LIN {X 0,Y 425.386,Z 292.31,A -85,B 0,C 180,E1 -9710.49,E2 -9710.49} C_VEL
LIN {X 0,Y 425.466,Z 292.296,A -85,B 0,C 180,E1 -9713.36,E2 -9713.36} C_VEL
LIN {X 0,Y 425.334,Z 292.312,A -85,B 0,C 180,E1 -9715.261,E2 -9715.261} C_VEL
LIN {X 0,Y 425.553,Z 292.292,A -85,B 0,C 180,E1 -9718.107,E2 -9718.107} C_VEL
LIN {X 0,Y 425.561,Z 292.291,A -85,B 0,C 180,E1 -9720,E2 -9720} C_VEL
LIN {X 0,Y 425.5,Z 292.291,A -85,B 0,C 180,E1 -9722.84,E2 -9722.84} C_VEL
LIN {X 0,Y 425.514,Z 292.294,A -85,B 0,C 180,E1 -9725.687,E2 -9725.687} C_VEL
LIN {X 0,Y 425.384,Z 292.306,A -85,B 0,C 180,E1 -9728.551,E2 -9728.551} C_VEL
LIN {X 0,Y 425.398,Z 292.305,A -85,B 0,C 180,E1 -9732.402,E2 -9732.402} C_VEL
LIN {X 0,Y 425.292,Z 292.321,A -85,B 0,C 180,E1 -9735.331,E2 -9735.331} C_VEL
LIN {X 0,Y 425.302,Z 292.316,A -85,B 0,C 180,E1 -9738.299,E2 -9738.299} C_VEL
LIN {X 0,Y 425.277,Z 292.324,A -85,B 0,C 180,E1 -9741.319,E2 -9741.319} C_VEL
LIN {X 0,Y 425.288,Z 292.318,A -85,B 0,C 180,E1 -9744.651,E2 -9744.651} C_VEL
LIN {X 0,Y 425.238,Z 292.328,A -85,B 0,C 180,E1 -9747.565,E2 -9747.565} C_VEL
LIN {X 0,Y 425.28,Z 292.321,A -85,B 0,C 180,E1 -9750.761,E2 -9750.761} C_VEL
LIN {X 0,Y 425.283,Z 292.318,A -85,B 0,C 180,E1 -9754.284,E2 -9754.284} C_VEL
LIN {X 0,Y 425.268,Z 292.321,A -85,B 0,C 180,E1 -9757.695,E2 -9757.695} C_VEL
LIN {X 0,Y 425.236,Z 292.326,A -85,B 0,C 180,E1 -9760.515,E2 -9760.515} C_VEL
LIN {X 0,Y 425.239,Z 292.326,A -85,B 0,C 180,E1 -9763.35,E2 -9763.35} C_VEL
LIN {X 0,Y 425.251,Z 292.323,A -85,B 0,C 180,E1 -9766.044,E2 -9766.044} C_VEL
LIN {X 0,Y 425.242,Z 292.329,A -85,B 0,C 180,E1 -9768.619,E2 -9768.619} C_VEL
LIN {X 0,Y 425.272,Z 292.323,A -85,B 0,C 180,E1 -9771.1,E2 -9771.1} C_VEL
LIN {X 0,Y 425.29,Z 292.325,A -85,B 0,C 180,E1 -9774.664,E2 -9774.664} C_VEL
LIN {X 0,Y 425.258,Z 292.323,A -85,B 0,C 180,E1 -9778.073,E2 -9778.073} C_VEL
LIN {X 0,Y 425.293,Z 292.317,A -85,B 0,C 180,E1 -9781.366,E2 -9781.366} C_VEL
LIN {X 0,Y 425.257,Z 292.329,A -85,B 0,C 180,E1 -9784.553,E2 -9784.553} C_VEL
LIN {X 0,Y 425.389,Z 292.538,A -85,B 0,C 180,E1 -9787.296,E2 -9787.296} C_VEL
LIN {X 0,Y 426.425,Z 299.768,A -85,B 0,C 180,E1 -9789.247,E2 -9789.247} C_VEL
LIN {X 0,Y 426.191,Z 307.575,A -85,B 0,C 180,E1 -9791.243,E2 -9791.243} C_VEL
LIN {X 0,Y 425.59,Z 319.286,A -85,B 0,C 180,E1 -9794.189,E2 -9794.189} C_VEL
LIN {X 0,Y 425.42,Z 323.878,A -85,B 0,C 180,E1 -9795.256,E2 -9795.256} C_VEL
LIN {X 0,Y 427.716,Z 338.164,A -85,B 0,C 180,E1 -9795.613,E2 -9795.613} C_VEL
LIN {X 0,Y 428.197,Z 343.55,A -85,B 0,C 180,E1 -9795.721,E2 -9795.721} C_VEL
LIN {X 0,Y 427.792,Z 399.196,A -85,B 0,C 180,E1 -9796.671,E2 -9796.671} C_VEL
LIN {X 0,Y 427.517,Z 408.492,A -85,B 0,C 180,E1 -9796.936,E2 -9796.936} C_VEL
LIN {X 0,Y 427.221,Z 418.151,A -85,B 0,C 180,E1 -9797.35,E2 -9797.35} C_VEL
LIN {X 0,Y 426.799,Z 427.305,A -85,B 0,C 180,E1 -9797.881,E2 -9797.881} C_VEL
LIN {X 0,Y 426.301,Z 438.098,A -85,B 0,C 180,E1 -9798.711,E2 -9798.711} C_VEL
LIN {X 0,Y 425.785,Z 447.393,A -85,B 0,C 180,E1 -9799.659,E2 -9799.659} C_VEL
LIN {X 0,Y 425.404,Z 454.053,A -85,B 0,C 180,E1 -9800.491,E2 -9800.491} C_VEL
LIN {X 0,Y 425.02,Z 460.372,A -85,B 0,C 180,E1 -9801.442,E2 -9801.442} C_VEL
LIN {X 0,Y 424.765,Z 465.622,A -85,B 0,C 180,E1 -9802.394,E2 -9802.394} C_VEL
LIN {X 0,Y 424.579,Z 469.999,A -85,B 0,C 180,E1 -9803.346,E2 -9803.346} C_VEL
LIN {X 0,Y 424.42,Z 473.64,A -85,B 0,C 180,E1 -9804.298,E2 -9804.298} C_VEL
LIN {X 0,Y 424.265,Z 476.628,A -85,B 0,C 180,E1 -9805.249,E2 -9805.249} C_VEL
LIN {X 0,Y 424.159,Z 478.944,A -85,B 0,C 180,E1 -9806.2,E2 -9806.2} C_VEL
LIN {X 0,Y 424.151,Z 480.684,A -85,B 0,C 180,E1 -9807.151,E2 -9807.151} C_VEL
LIN {X 0,Y 424.129,Z 481.93,A -85,B 0,C 180,E1 -9808.101,E2 -9808.101} C_VEL
LIN {X 0,Y 424.067,Z 482.706,A -85,B 0,C 180,E1 -9809.05,E2 -9809.05} C_VEL
LIN {X 0,Y 424.039,Z 483,A -85,B 0,C 180,E1 -9810,E2 -9810} C_VEL
LIN {X 0,Y 424.067,Z 482.704,A -85,B 0,C 180,E1 -9810.95,E2 -9810.95} C_VEL
LIN {X 0,Y 424.129,Z 481.925,A -85,B 0,C 180,E1 -9811.899,E2 -9811.899} C_VEL
LIN {X 0,Y 424.15,Z 480.675,A -85,B 0,C 180,E1 -9812.849,E2 -9812.849} C_VEL
LIN {X 0,Y 424.198,Z 477.78,A -85,B 0,C 180,E1 -9814.276,E2 -9814.276} C_VEL
LIN {X 0,Y 424.364,Z 475.142,A -85,B 0,C 180,E1 -9815.226,E2 -9815.226} C_VEL
LIN {X 0,Y 424.496,Z 471.301,A -85,B 0,C 180,E1 -9816.324,E2 -9816.324} C_VEL
LIN {X 0,Y 424.759,Z 465.592,A -85,B 0,C 180,E1 -9817.606,E2 -9817.606} C_VEL
LIN {X 0,Y 425.105,Z 458.923,A -85,B 0,C 180,E1 -9818.796,E2 -9818.796} C_VEL
LIN {X 0,Y 425.61,Z 450.418,A -85,B 0,C 180,E1 -9819.984,E2 -9819.984} C_VEL
LIN {X 0,Y 426.102,Z 441.738,A -85,B 0,C 180,E1 -9820.934,E2 -9820.934} C_VEL
LIN {X 0,Y 426.555,Z 433.692,A -85,B 0,C 180,E1 -9821.644,E2 -9821.644} C_VEL
LIN {X 0,Y 426.913,Z 425.352,A -85,B 0,C 180,E1 -9822.237,E2 -9822.237} C_VEL
LIN {X 0,Y 427.243,Z 416.837,A -85,B 0,C 180,E1 -9822.71,E2 -9822.71} C_VEL
LIN {X 0,Y 427.565,Z 406.683,A -85,B 0,C 180,E1 -9823.123,E2 -9823.123} C_VEL
LIN {X 0,Y 427.827,Z 394.605,A -85,B 0,C 180,E1 -9823.422,E2 -9823.422} C_VEL
LIN {X 0,Y 428.101,Z 340.832,A -85,B 0,C 180,E1 -9824.323,E2 -9824.323} C_VEL
LIN {X 0,Y 425.441,Z 324.039,A -85,B 0,C 180,E1 -9824.725,E2 -9824.725} C_VEL
LIN {X 0,Y 425.418,Z 322.288,A -85,B 0,C 180,E1 -9825.057,E2 -9825.057} C_VEL
LIN {X 0,Y 425.958,Z 311.453,A -85,B 0,C 180,E1 -9827.772,E2 -9827.772} C_VEL
LIN {X 0,Y 426.464,Z 301.692,A -85,B 0,C 180,E1 -9830.247,E2 -9830.247} C_VEL
LIN {X 0,Y 425.949,Z 295.836,A -85,B 0,C 180,E1 -9831.792,E2 -9831.792} C_VEL
LIN {X 0,Y 425.345,Z 292.395,A -85,B 0,C 180,E1 -9832.777,E2 -9832.777} C_VEL
LIN {X 0,Y 425.257,Z 292.329,A -85,B 0,C 180,E1 -9835.447,E2 -9835.447} C_VEL
LIN {X 0,Y 425.303,Z 292.317,A -85,B 0,C 180,E1 -9838.859,E2 -9838.859} C_VEL
LIN {X 0,Y 425.258,Z 292.323,A -85,B 0,C 180,E1 -9841.927,E2 -9841.927} C_VEL
LIN {X 0,Y 425.29,Z 292.325,A -85,B 0,C 180,E1 -9845.336,E2 -9845.336} C_VEL
LIN {X 0,Y 425.275,Z 292.322,A -85,B 0,C 180,E1 -9848.9,E2 -9848.9} C_VEL
LIN {X 0,Y 425.25,Z 292.324,A -85,B 0,C 180,E1 -9852.655,E2 -9852.655} C_VEL
LIN {X 0,Y 425.278,Z 292.324,A -85,B 0,C 180,E1 -9855.283,E2 -9855.283} C_VEL
LIN {X 0,Y 425.24,Z 292.326,A -85,B 0,C 180,E1 -9858.617,E2 -9858.617} C_VEL
LIN {X 0,Y 425.273,Z 292.325,A -85,B 0,C 180,E1 -9861.099,E2 -9861.099} C_VEL
LIN {X 0,Y 425.286,Z 292.323,A -85,B 0,C 180,E1 -9864.663,E2 -9864.663} C_VEL
LIN {X 0,Y 425.252,Z 292.323,A -85,B 0,C 180,E1 -9868.072,E2 -9868.072} C_VEL
LIN {X 0,Y 425.287,Z 292.319,A -85,B 0,C 180,E1 -9871.365,E2 -9871.365} C_VEL
LIN {X 0,Y 425.25,Z 292.329,A -85,B 0,C 180,E1 -9874.552,E2 -9874.552} C_VEL
LIN {X 0,Y 425.282,Z 292.319,A -85,B 0,C 180,E1 -9877.73,E2 -9877.73} C_VEL
LIN {X 0,Y 425.35,Z 292.315,A -85,B 0,C 180,E1 -9880.704,E2 -9880.704} C_VEL
LIN {X 0,Y 425.308,Z 292.316,A -85,B 0,C 180,E1 -9883.685,E2 -9883.685} C_VEL
LIN {X 0,Y 425.384,Z 292.306,A -85,B 0,C 180,E1 -9887.097,E2 -9887.097} C_VEL
LIN {X 0,Y 425.383,Z 292.31,A -85,B 0,C 180,E1 -9890.49,E2 -9890.49} C_VEL
LIN {X 0,Y 425.466,Z 292.296,A -85,B 0,C 180,E1 -9893.36,E2 -9893.36} C_VEL
LIN {X 0,Y 425.334,Z 292.312,A -85,B 0,C 180,E1 -9895.261,E2 -9895.261} C_VEL
LIN {X 0,Y 425.553,Z 292.292,A -85,B 0,C 180,E1 -9898.107,E2 -9898.107} C_VEL
LIN {X 0,Y 425.561,Z 292.291,A -85,B 0,C 180,E1 -9900,E2 -9900} C_VEL
LIN {X 0,Y 425.5,Z 292.291,A -85,B 0,C 180,E1 -9902.84,E2 -9902.84} C_VEL
LIN {X 0,Y 425.466,Z 292.296,A -85,B 0,C 180,E1 -9906.457,E2 -9906.457} C_VEL
LIN {X 0,Y 425.369,Z 292.312,A -85,B 0,C 180,E1 -9909.51,E2 -9909.51} C_VEL
LIN {X 0,Y 425.383,Z 292.306,A -85,B 0,C 180,E1 -9912.903,E2 -9912.903} C_VEL
LIN {X 0,Y 425.304,Z 292.316,A -85,B 0,C 180,E1 -9916.583,E2 -9916.583} C_VEL
LIN {X 0,Y 425.318,Z 292.32,A -85,B 0,C 180,E1 -9919.635,E2 -9919.635} C_VEL
LIN {X 0,Y 425.276,Z 292.319,A -85,B 0,C 180,E1 -9922.339,E2 -9922.339} C_VEL
LIN {X 0,Y 425.25,Z 292.329,A -85,B 0,C 180,E1 -9925.448,E2 -9925.448} C_VEL
LIN {X 0,Y 425.291,Z 292.32,A -85,B 0,C 180,E1 -9928.859,E2 -9928.859} C_VEL
LIN {X 0,Y 425.245,Z 292.324,A -85,B 0,C 180,E1 -9931.929,E2 -9931.929} C_VEL
LIN {X 0,Y 425.287,Z 292.323,A -85,B 0,C 180,E1 -9935.337,E2 -9935.337} C_VEL
LIN {X 0,Y 425.271,Z 292.325,A -85,B 0,C 180,E1 -9938.902,E2 -9938.902} C_VEL
LIN {X 0,Y 425.25,Z 292.326,A -85,B 0,C 180,E1 -9942.656,E2 -9942.656} C_VEL
LIN {X 0,Y 425.28,Z 292.322,A -85,B 0,C 180,E1 -9945.284,E2 -9945.284} C_VEL
LIN {X 0,Y 425.243,Z 292.328,A -85,B 0,C 180,E1 -9948.619,E2 -9948.619} C_VEL
LIN {X 0,Y 425.273,Z 292.323,A -85,B 0,C 180,E1 -9951.1,E2 -9951.1} C_VEL
LIN {X 0,Y 425.291,Z 292.325,A -85,B 0,C 180,E1 -9954.664,E2 -9954.664} C_VEL
LIN {X 0,Y 425.25,Z 292.324,A -85,B 0,C 180,E1 -9958.073,E2 -9958.073} C_VEL
LIN {X 0,Y 425.289,Z 292.318,A -85,B 0,C 180,E1 -9961.366,E2 -9961.366} C_VEL
LIN {X 0,Y 425.258,Z 292.329,A -85,B 0,C 180,E1 -9964.553,E2 -9964.553} C_VEL
LIN {X 0,Y 425.379,Z 292.495,A -85,B 0,C 180,E1 -9967.331,E2 -9967.331} C_VEL
LIN {X 0,Y 426.384,Z 299.567,A -85,B 0,C 180,E1 -9969.245,E2 -9969.245} C_VEL
LIN {X 0,Y 426.293,Z 305.422,A -85,B 0,C 180,E1 -9970.748,E2 -9970.748} C_VEL
LIN {X 0,Y 425.592,Z 319.083,A -85,B 0,C 180,E1 -9974.189,E2 -9974.189} C_VEL
LIN {X 0,Y 425.407,Z 323.763,A -85,B 0,C 180,E1 -9975.295,E2 -9975.295} C_VEL
LIN {X 0,Y 426.275,Z 329.311,A -85,B 0,C 180,E1 -9975.463,E2 -9975.463} C_VEL
LIN {X 0,Y 428.127,Z 342.177,A -85,B 0,C 180,E1 -9975.746,E2 -9975.746} C_VEL
LIN {X 0,Y 427.793,Z 399.7,A -85,B 0,C 180,E1 -9976.734,E2 -9976.734} C_VEL
LIN {X 0,Y 427.51,Z 408.771,A -85,B 0,C 180,E1 -9976.997,E2 -9976.997} C_VEL
LIN {X 0,Y 427.189,Z 418.355,A -85,B 0,C 180,E1 -9977.41,E2 -9977.41} C_VEL
LIN {X 0,Y 426.755,Z 428.398,A -85,B 0,C 180,E1 -9978,E2 -9978} C_VEL
LIN {X 0,Y 426.307,Z 438.818,A -85,B 0,C 180,E1 -9978.831,E2 -9978.831} C_VEL
LIN {X 0,Y 425.832,Z 446.973,A -85,B 0,C 180,E1 -9979.661,E2 -9979.661} C_VEL
LIN {X 0,Y 425.418,Z 453.702,A -85,B 0,C 180,E1 -9980.491,E2 -9980.491} C_VEL
LIN {X 0,Y 425.027,Z 460.074,A -85,B 0,C 180,E1 -9981.442,E2 -9981.442} C_VEL
LIN {X 0,Y 424.982,Z 461.255,A -85,B 0,C 180,E1 -9981.64,E2 -9981.64} C_VEL
LIN {X 0,Y 424.187,Z 464.868,A -85,B 0,C 180,E1 -9982.267,E2 -9982.267} C_VEL
LIN {X 0,Y 421.107,Z 470.148,A -85,B 0,C 180,E1 -9983.327,E2 -9983.327} C_VEL
LIN {X 0,Y 418.008,Z 474.51,A -85,B 0,C 180,E1 -9984.472,E2 -9984.472} C_VEL
LIN {X 0,Y 417.196,Z 476.627,A -85,B 0,C 180,E1 -9985.224,E2 -9985.224} C_VEL
LIN {X 0,Y 417.074,Z 478.823,A -85,B 0,C 180,E1 -9986.135,E2 -9986.135} C_VEL
LIN {X 0,Y 417.051,Z 480.599,A -85,B 0,C 180,E1 -9987.102,E2 -9987.102} C_VEL
LIN {X 0,Y 417.058,Z 481.88,A -85,B 0,C 180,E1 -9988.069,E2 -9988.069} C_VEL
LIN {X 0,Y 416.991,Z 482.689,A -85,B 0,C 180,E1 -9989.034,E2 -9989.034} C_VEL
LIN {X 0,Y 416.962,Z 482.998,A -85,B 0,C 180,E1 -9990,E2 -9990} C_VEL
LIN {X 0,Y 416.991,Z 482.721,A -85,B 0,C 180,E1 -9990.966,E2 -9990.966} C_VEL
LIN {X 0,Y 417.037,Z 481.976,A -85,B 0,C 180,E1 -9991.931,E2 -9991.931} C_VEL
LIN {X 0,Y 417.041,Z 480.76,A -85,B 0,C 180,E1 -9992.898,E2 -9992.898} C_VEL
LIN {X 0,Y 417.122,Z 477.9,A -85,B 0,C 180,E1 -9994.348,E2 -9994.348} C_VEL
LIN {X 0,Y 417.267,Z 475.299,A -85,B 0,C 180,E1 -9995.315,E2 -9995.315} C_VEL
LIN {X 0,Y 417.521,Z 470.177,A -85,B 0,C 180,E1 -9996.767,E2 -9996.767} C_VEL
LIN {X 0,Y 417.75,Z 464.668,A -85,B 0,C 180,E1 -9997.978,E2 -9997.978} C_VEL
LIN {X 0,Y 418.174,Z 457.753,A -85,B 0,C 180,E1 -9999.187,E2 -9999.187} C_VEL
LIN {X 0,Y 418.673,Z 449.813,A -85,B 0,C 180,E1 -10000.274,E2 -10000.274} C_VEL
LIN {X 0,Y 419.102,Z 442.243,A -85,B 0,C 180,E1 -10001.119,E2 -10001.119} C_VEL
LIN {X 0,Y 419.568,Z 434.311,A -85,B 0,C 180,E1 -10001.841,E2 -10001.841} C_VEL
LIN {X 0,Y 419.963,Z 426.124,A -85,B 0,C 180,E1 -10002.442,E2 -10002.442} C_VEL
LIN {X 0,Y 420.362,Z 417.834,A -85,B 0,C 180,E1 -10002.921,E2 -10002.921} C_VEL
LIN {X 0,Y 420.621,Z 408.887,A -85,B 0,C 180,E1 -10003.312,E2 -10003.312} C_VEL
LIN {X 0,Y 420.872,Z 399.665,A -85,B 0,C 180,E1 -10003.586,E2 -10003.586} C_VEL
LIN {X 0,Y 421.13,Z 340.835,A -85,B 0,C 180,E1 -10004.616,E2 -10004.616} C_VEL
LIN {X 0,Y 418.444,Z 324.13,A -85,B 0,C 180,E1 -10005.027,E2 -10005.027} C_VEL
LIN {X 0,Y 418.392,Z 323.498,A -85,B 0,C 180,E1 -10005.091,E2 -10005.091} C_VEL
LIN {X 0,Y 419.004,Z 311.653,A -85,B 0,C 180,E1 -10008.077,E2 -10008.077} C_VEL
LIN {X 0,Y 419.454,Z 301.892,A -85,B 0,C 180,E1 -10010.6,E2 -10010.6} C_VEL
LIN {X 0,Y 418.555,Z 294.691,A -85,B 0,C 180,E1 -10012.555,E2 -10012.555} C_VEL
LIN {X 0,Y 418.315,Z 293.276,A -85,B 0,C 180,E1 -10012.992,E2 -10012.992} C_VEL
LIN {X 0,Y 418.217,Z 293.203,A -85,B 0,C 180,E1 -10015.907,E2 -10015.907} C_VEL
LIN {X 0,Y 418.257,Z 293.196,A -85,B 0,C 180,E1 -10019.162,E2 -10019.162} C_VEL
LIN {X 0,Y 418.249,Z 293.196,A -85,B 0,C 180,E1 -10022.842,E2 -10022.842} C_VEL
LIN {X 0,Y 418.24,Z 293.196,A -85,B 0,C 180,E1 -10026.237,E2 -10026.237} C_VEL
LIN {X 0,Y 418.196,Z 293.204,A -85,B 0,C 180,E1 -10029.687,E2 -10029.687} C_VEL
LIN {X 0,Y 418.203,Z 293.2,A -85,B 0,C 180,E1 -10032.317,E2 -10032.317} C_VEL
LIN {X 0,Y 418.231,Z 293.204,A -85,B 0,C 180,E1 -10035.108,E2 -10035.108} C_VEL
LIN {X 0,Y 418.213,Z 293.2,A -85,B 0,C 180,E1 -10037.763,E2 -10037.763} C_VEL
LIN {X 0,Y 418.233,Z 293.198,A -85,B 0,C 180,E1 -10041.556,E2 -10041.556} C_VEL
LIN {X 0,Y 418.243,Z 293.199,A -85,B 0,C 180,E1 -10045.157,E2 -10045.157} C_VEL
LIN {X 0,Y 418.235,Z 293.197,A -85,B 0,C 180,E1 -10047.471,E2 -10047.471} C_VEL
LIN {X 0,Y 418.251,Z 293.2,A -85,B 0,C 180,E1 -10050.897,E2 -10050.897} C_VEL
LIN {X 0,Y 418.21,Z 293.201,A -85,B 0,C 180,E1 -10054.092,E2 -10054.092} C_VEL
LIN {X 0,Y 418.218,Z 293.199,A -85,B 0,C 180,E1 -10057.263,E2 -10057.263} C_VEL
LIN {X 0,Y 418.273,Z 293.197,A -85,B 0,C 180,E1 -10060.364,E2 -10060.364} C_VEL
LIN {X 0,Y 418.27,Z 293.192,A -85,B 0,C 180,E1 -10063.403,E2 -10063.403} C_VEL
LIN {X 0,Y 418.337,Z 293.184,A -85,B 0,C 180,E1 -10066.999,E2 -10066.999} C_VEL
LIN {X 0,Y 418.327,Z 293.191,A -85,B 0,C 180,E1 -10070.328,E2 -10070.328} C_VEL
LIN {X 0,Y 418.431,Z 293.172,A -85,B 0,C 180,E1 -10073.248,E2 -10073.248} C_VEL
LIN {X 0,Y 418.306,Z 293.187,A -85,B 0,C 180,E1 -10075.181,E2 -10075.181} C_VEL
LIN {X 0,Y 418.522,Z 293.168,A -85,B 0,C 180,E1 -10078.075,E2 -10078.075} C_VEL
LIN {X 0,Y 418.395,Z 293.176,A -85,B 0,C 180,E1 -10080.962,E2 -10080.962} C_VEL
LIN {X 0,Y 418.457,Z 293.169,A -85,B 0,C 180,E1 -10082.888,E2 -10082.888} C_VEL
LIN {X 0,Y 418.472,Z 293.173,A -85,B 0,C 180,E1 -10085.783,E2 -10085.783} C_VEL
LIN {X 0,Y 418.356,Z 293.181,A -85,B 0,C 180,E1 -10088.696,E2 -10088.696} C_VEL
LIN {X 0,Y 418.343,Z 293.183,A -85,B 0,C 180,E1 -10092.615,E2 -10092.615} C_VEL
LIN {X 0,Y 418.241,Z 293.203,A -85,B 0,C 180,E1 -10095.596,E2 -10095.596} C_VEL
LIN {X 0,Y 418.259,Z 293.193,A -85,B 0,C 180,E1 -10098.618,E2 -10098.618} C_VEL
LIN {X 0,Y 418.22,Z 293.203,A -85,B 0,C 180,E1 -10101.697,E2 -10101.697} C_VEL
LIN {X 0,Y 418.235,Z 293.198,A -85,B 0,C 180,E1 -10104.853,E2 -10104.853} C_VEL
LIN {X 0,Y 418.198,Z 293.201,A -85,B 0,C 180,E1 -10108.07,E2 -10108.07} C_VEL
LIN {X 0,Y 418.229,Z 293.202,A -85,B 0,C 180,E1 -10111.019,E2 -10111.019} C_VEL
LIN {X 0,Y 418.224,Z 293.2,A -85,B 0,C 180,E1 -10113.679,E2 -10113.679} C_VEL
LIN {X 0,Y 418.23,Z 293.203,A -85,B 0,C 180,E1 -10117.225,E2 -10117.225} C_VEL
LIN {X 0,Y 418.2,Z 293.206,A -85,B 0,C 180,E1 -10120.868,E2 -10120.868} C_VEL
LIN {X 0,Y 418.196,Z 293.202,A -85,B 0,C 180,E1 -10123.729,E2 -10123.729} C_VEL
LIN {X 0,Y 418.193,Z 293.204,A -85,B 0,C 180,E1 -10126.448,E2 -10126.448} C_VEL
LIN {X 0,Y 418.201,Z 293.204,A -85,B 0,C 180,E1 -10129.134,E2 -10129.134} C_VEL
LIN {X 0,Y 418.231,Z 293.203,A -85,B 0,C 180,E1 -10132.776,E2 -10132.776} C_VEL
LIN {X 0,Y 418.228,Z 293.201,A -85,B 0,C 180,E1 -10136.322,E2 -10136.322} C_VEL
LIN {X 0,Y 418.235,Z 293.197,A -85,B 0,C 180,E1 -10139.728,E2 -10139.728} C_VEL
LIN {X 0,Y 418.207,Z 293.201,A -85,B 0,C 180,E1 -10143.017,E2 -10143.017} C_VEL
LIN {X 0,Y 418.279,Z 293.178,A -85,B 0,C 180,E1 -10146.219,E2 -10146.219} C_VEL
LIN {X 0,Y 418.341,Z 293.45,A -85,B 0,C 180,E1 -10147.14,E2 -10147.14} C_VEL
LIN {X 0,Y 419.345,Z 299.769,A -85,B 0,C 180,E1 -10148.88,E2 -10148.88} C_VEL
LIN {X 0,Y 419.366,Z 305.625,A -85,B 0,C 180,E1 -10150.417,E2 -10150.417} C_VEL
LIN {X 0,Y 418.629,Z 319.287,A -85,B 0,C 180,E1 -10153.919,E2 -10153.919} C_VEL
LIN {X 0,Y 418.424,Z 323.88,A -85,B 0,C 180,E1 -10155.004,E2 -10155.004} C_VEL
LIN {X 0,Y 420.761,Z 338.486,A -85,B 0,C 180,E1 -10155.375,E2 -10155.375} C_VEL
LIN {X 0,Y 421.338,Z 343.569,A -85,B 0,C 180,E1 -10155.483,E2 -10155.483} C_VEL
LIN {X 0,Y 420.903,Z 399.263,A -85,B 0,C 180,E1 -10156.45,E2 -10156.45} C_VEL
LIN {X 0,Y 420.618,Z 408.501,A -85,B 0,C 180,E1 -10156.718,E2 -10156.718} C_VEL
LIN {X 0,Y 420.344,Z 416.948,A -85,B 0,C 180,E1 -10157.078,E2 -10157.078} C_VEL
LIN {X 0,Y 419.962,Z 425.438,A -85,B 0,C 180,E1 -10157.558,E2 -10157.558} C_VEL
LIN {X 0,Y 419.586,Z 433.761,A -85,B 0,C 180,E1 -10158.16,E2 -10158.16} C_VEL
LIN {X 0,Y 419.15,Z 441.791,A -85,B 0,C 180,E1 -10158.883,E2 -10158.883} C_VEL
LIN {X 0,Y 418.597,Z 450.457,A -85,B 0,C 180,E1 -10159.847,E2 -10159.847} C_VEL
LIN {X 0,Y 418.086,Z 458.955,A -85,B 0,C 180,E1 -10161.055,E2 -10161.055} C_VEL
LIN {X 0,Y 417.706,Z 465.624,A -85,B 0,C 180,E1 -10162.265,E2 -10162.265} C_VEL
LIN {X 0,Y 417.509,Z 470.232,A -85,B 0,C 180,E1 -10163.292,E2 -10163.292} C_VEL
LIN {X 0,Y 417.286,Z 475.158,A -85,B 0,C 180,E1 -10164.685,E2 -10164.685} C_VEL
LIN {X 0,Y 417.072,Z 478.944,A -85,B 0,C 180,E1 -10166.135,E2 -10166.135} C_VEL
LIN {X 0,Y 417.05,Z 480.684,A -85,B 0,C 180,E1 -10167.102,E2 -10167.102} C_VEL
LIN {X 0,Y 417.057,Z 481.931,A -85,B 0,C 180,E1 -10168.069,E2 -10168.069} C_VEL
LIN {X 0,Y 416.991,Z 482.706,A -85,B 0,C 180,E1 -10169.034,E2 -10169.034} C_VEL
LIN {X 0,Y 416.961,Z 483,A -85,B 0,C 180,E1 -10170,E2 -10170} C_VEL
LIN {X 0,Y 416.991,Z 482.704,A -85,B 0,C 180,E1 -10170.966,E2 -10170.966} C_VEL
LIN {X 0,Y 417.057,Z 481.925,A -85,B 0,C 180,E1 -10171.931,E2 -10171.931} C_VEL
LIN {X 0,Y 417.049,Z 480.674,A -85,B 0,C 180,E1 -10172.898,E2 -10172.898} C_VEL
LIN {X 0,Y 417.123,Z 477.78,A -85,B 0,C 180,E1 -10174.348,E2 -10174.348} C_VEL
LIN {X 0,Y 417.285,Z 475.141,A -85,B 0,C 180,E1 -10175.315,E2 -10175.315} C_VEL
LIN {X 0,Y 417.519,Z 469.975,A -85,B 0,C 180,E1 -10176.767,E2 -10176.767} C_VEL
LIN {X 0,Y 417.836,Z 463.167,A -85,B 0,C 180,E1 -10178.22,E2 -10178.22} C_VEL
LIN {X 0,Y 418.273,Z 455.72,A -85,B 0,C 180,E1 -10179.429,E2 -10179.429} C_VEL
LIN {X 0,Y 418.745,Z 448.374,A -85,B 0,C 180,E1 -10180.394,E2 -10180.394} C_VEL
LIN {X 0,Y 419.207,Z 440.505,A -85,B 0,C 180,E1 -10181.238,E2 -10181.238} C_VEL
LIN {X 0,Y 419.666,Z 432.187,A -85,B 0,C 180,E1 -10181.96,E2 -10181.96} C_VEL
LIN {X 0,Y 420.163,Z 421.563,A -85,B 0,C 180,E1 -10182.682,E2 -10182.682} C_VEL
LIN {X 0,Y 420.551,Z 410,A -85,B 0,C 180,E1 -10183.222,E2 -10183.222} C_VEL
LIN {X 0,Y 420.85,Z 400.32,A -85,B 0,C 180,E1 -10183.52,E2 -10183.52} C_VEL
LIN {X 0,Y 421.152,Z 340.97,A -85,B 0,C 180,E1 -10184.562,E2 -10184.562} C_VEL
LIN {X 0,Y 418.462,Z 324.288,A -85,B 0,C 180,E1 -10184.963,E2 -10184.963} C_VEL
LIN {X 0,Y 418.388,Z 322.846,A -85,B 0,C 180,E1 -10185.179,E2 -10185.179} C_VEL
LIN {X 0,Y 419.003,Z 311.452,A -85,B 0,C 180,E1 -10188.077,E2 -10188.077} C_VEL
LIN {X 0,Y 419.477,Z 303.049,A -85,B 0,C 180,E1 -10190.243,E2 -10190.243} C_VEL
LIN {X 0,Y 419.071,Z 297.786,A -85,B 0,C 180,E1 -10191.65,E2 -10191.65} C_VEL
LIN {X 0,Y 418.328,Z 293.282,A -85,B 0,C 180,E1 -10192.926,E2 -10192.926} C_VEL
LIN {X 0,Y 418.216,Z 293.202,A -85,B 0,C 180,E1 -10195.907,E2 -10195.907} C_VEL
LIN {X 0,Y 418.255,Z 293.197,A -85,B 0,C 180,E1 -10199.162,E2 -10199.162} C_VEL
LIN {X 0,Y 418.247,Z 293.196,A -85,B 0,C 180,E1 -10202.842,E2 -10202.842} C_VEL
LIN {X 0,Y 418.238,Z 293.196,A -85,B 0,C 180,E1 -10206.237,E2 -10206.237} C_VEL
LIN {X 0,Y 418.195,Z 293.204,A -85,B 0,C 180,E1 -10209.687,E2 -10209.687} C_VEL
LIN {X 0,Y 418.202,Z 293.201,A -85,B 0,C 180,E1 -10212.317,E2 -10212.317} C_VEL
LIN {X 0,Y 418.23,Z 293.204,A -85,B 0,C 180,E1 -10215.108,E2 -10215.108} C_VEL
LIN {X 0,Y 418.212,Z 293.2,A -85,B 0,C 180,E1 -10217.763,E2 -10217.763} C_VEL
LIN {X 0,Y 418.23,Z 293.198,A -85,B 0,C 180,E1 -10221.556,E2 -10221.556} C_VEL
LIN {X 0,Y 418.242,Z 293.199,A -85,B 0,C 180,E1 -10225.158,E2 -10225.158} C_VEL
LIN {X 0,Y 418.234,Z 293.197,A -85,B 0,C 180,E1 -10227.471,E2 -10227.471} C_VEL
LIN {X 0,Y 418.251,Z 293.2,A -85,B 0,C 180,E1 -10230.898,E2 -10230.898} C_VEL
LIN {X 0,Y 418.209,Z 293.201,A -85,B 0,C 180,E1 -10234.092,E2 -10234.092} C_VEL
LIN {X 0,Y 418.217,Z 293.199,A -85,B 0,C 180,E1 -10237.263,E2 -10237.263} C_VEL
LIN {X 0,Y 418.273,Z 293.197,A -85,B 0,C 180,E1 -10240.364,E2 -10240.364} C_VEL
LIN {X 0,Y 418.27,Z 293.192,A -85,B 0,C 180,E1 -10243.403,E2 -10243.403} C_VEL
LIN {X 0,Y 418.337,Z 293.184,A -85,B 0,C 180,E1 -10247,E2 -10247} C_VEL
LIN {X 0,Y 418.324,Z 293.192,A -85,B 0,C 180,E1 -10250.328,E2 -10250.328} C_VEL
LIN {X 0,Y 418.431,Z 293.172,A -85,B 0,C 180,E1 -10253.248,E2 -10253.248} C_VEL
LIN {X 0,Y 418.306,Z 293.187,A -85,B 0,C 180,E1 -10255.181,E2 -10255.181} C_VEL
LIN {X 0,Y 418.522,Z 293.168,A -85,B 0,C 180,E1 -10258.075,E2 -10258.075} C_VEL
LIN {X 0,Y 418.395,Z 293.176,A -85,B 0,C 180,E1 -10260.963,E2 -10260.963} C_VEL
LIN {X 0,Y 418.457,Z 293.169,A -85,B 0,C 180,E1 -10262.888,E2 -10262.888} C_VEL
LIN {X 0,Y 418.431,Z 293.172,A -85,B 0,C 180,E1 -10266.454,E2 -10266.454} C_VEL
LIN {X 0,Y 418.356,Z 293.181,A -85,B 0,C 180,E1 -10268.696,E2 -10268.696} C_VEL
LIN {X 0,Y 418.343,Z 293.183,A -85,B 0,C 180,E1 -10272.615,E2 -10272.615} C_VEL
LIN {X 0,Y 418.239,Z 293.203,A -85,B 0,C 180,E1 -10275.597,E2 -10275.597} C_VEL
LIN {X 0,Y 418.254,Z 293.194,A -85,B 0,C 180,E1 -10278.618,E2 -10278.618} C_VEL
LIN {X 0,Y 418.221,Z 293.203,A -85,B 0,C 180,E1 -10281.697,E2 -10281.697} C_VEL
LIN {X 0,Y 418.236,Z 293.198,A -85,B 0,C 180,E1 -10284.853,E2 -10284.853} C_VEL
LIN {X 0,Y 418.198,Z 293.201,A -85,B 0,C 180,E1 -10288.07,E2 -10288.07} C_VEL
LIN {X 0,Y 418.228,Z 293.201,A -85,B 0,C 180,E1 -10291.019,E2 -10291.019} C_VEL
LIN {X 0,Y 418.224,Z 293.2,A -85,B 0,C 180,E1 -10293.679,E2 -10293.679} C_VEL
LIN {X 0,Y 418.229,Z 293.203,A -85,B 0,C 180,E1 -10297.225,E2 -10297.225} C_VEL
LIN {X 0,Y 418.201,Z 293.206,A -85,B 0,C 180,E1 -10300.868,E2 -10300.868} C_VEL
LIN {X 0,Y 418.197,Z 293.201,A -85,B 0,C 180,E1 -10303.729,E2 -10303.729} C_VEL
LIN {X 0,Y 418.194,Z 293.204,A -85,B 0,C 180,E1 -10306.448,E2 -10306.448} C_VEL
LIN {X 0,Y 418.202,Z 293.204,A -85,B 0,C 180,E1 -10309.134,E2 -10309.134} C_VEL
LIN {X 0,Y 418.232,Z 293.204,A -85,B 0,C 180,E1 -10312.776,E2 -10312.776} C_VEL
LIN {X 0,Y 418.229,Z 293.2,A -85,B 0,C 180,E1 -10316.322,E2 -10316.322} C_VEL
LIN {X 0,Y 418.231,Z 293.197,A -85,B 0,C 180,E1 -10319.728,E2 -10319.728} C_VEL
LIN {X 0,Y 418.206,Z 293.202,A -85,B 0,C 180,E1 -10323.017,E2 -10323.017} C_VEL
LIN {X 0,Y 418.274,Z 293.18,A -85,B 0,C 180,E1 -10326.219,E2 -10326.219} C_VEL
LIN {X 0,Y 418.316,Z 293.316,A -85,B 0,C 180,E1 -10327.138,E2 -10327.138} C_VEL
LIN {X 0,Y 419.286,Z 299.569,A -85,B 0,C 180,E1 -10328.877,E2 -10328.877} C_VEL
LIN {X 0,Y 419.367,Z 305.424,A -85,B 0,C 180,E1 -10330.418,E2 -10330.418} C_VEL
LIN {X 0,Y 418.631,Z 319.085,A -85,B 0,C 180,E1 -10333.919,E2 -10333.919} C_VEL
LIN {X 0,Y 418.411,Z 323.766,A -85,B 0,C 180,E1 -10335.043,E2 -10335.043} C_VEL
LIN {X 0,Y 419.339,Z 329.658,A -85,B 0,C 180,E1 -10335.223,E2 -10335.223} C_VEL
LIN {X 0,Y 421.271,Z 343.165,A -85,B 0,C 180,E1 -10335.525,E2 -10335.525} C_VEL
LIN {X 0,Y 420.898,Z 399.719,A -85,B 0,C 180,E1 -10336.512,E2 -10336.512} C_VEL
LIN {X 0,Y 420.617,Z 408.783,A -85,B 0,C 180,E1 -10336.78,E2 -10336.78} C_VEL
LIN {X 0,Y 420.253,Z 418.364,A -85,B 0,C 180,E1 -10337.198,E2 -10337.198} C_VEL
LIN {X 0,Y 419.832,Z 428.404,A -85,B 0,C 180,E1 -10337.799,E2 -10337.799} C_VEL
LIN {X 0,Y 419.346,Z 438.823,A -85,B 0,C 180,E1 -10338.643,E2 -10338.643} C_VEL
LIN {X 0,Y 418.842,Z 446.977,A -85,B 0,C 180,E1 -10339.486,E2 -10339.486} C_VEL
LIN {X 0,Y 418.426,Z 453.705,A -85,B 0,C 180,E1 -10340.331,E2 -10340.331} C_VEL
LIN {X 0,Y 418.007,Z 460.077,A -85,B 0,C 180,E1 -10341.297,E2 -10341.297} C_VEL
LIN {X 0,Y 417.681,Z 466.547,A -85,B 0,C 180,E1 -10342.507,E2 -10342.507} C_VEL
LIN {X 0,Y 417.397,Z 471.693,A -85,B 0,C 180,E1 -10343.712,E2 -10343.712} C_VEL
LIN {X 0,Y 417.196,Z 476.627,A -85,B 0,C 180,E1 -10345.224,E2 -10345.224} C_VEL
LIN {X 0,Y 416.422,Z 478.533,A -85,B 0,C 180,E1 -10345.992,E2 -10345.992} C_VEL
LIN {X 0,Y 413.477,Z 480.901,A -85,B 0,C 180,E1 -10347.259,E2 -10347.259} C_VEL
LIN {X 0,Y 411.04,Z 482.16,A -85,B 0,C 180,E1 -10348.298,E2 -10348.298} C_VEL
LIN {X 0,Y 409.985,Z 482.73,A -85,B 0,C 180,E1 -10349.11,E2 -10349.11} C_VEL
LIN {X 0,Y 409.892,Z 482.805,A -85,B 0,C 180,E1 -10349.385,E2 -10349.385} C_VEL
LIN {X 0,Y 409.886,Z 482.998,A -85,B 0,C 180,E1 -10350,E2 -10350} C_VEL
LIN {X 0,Y 409.917,Z 482.721,A -85,B 0,C 180,E1 -10350.982,E2 -10350.982} C_VEL
LIN {X 0,Y 409.949,Z 481.975,A -85,B 0,C 180,E1 -10351.965,E2 -10351.965} C_VEL
LIN {X 0,Y 409.941,Z 480.759,A -85,B 0,C 180,E1 -10352.948,E2 -10352.948} C_VEL
LIN {X 0,Y 410.052,Z 477.899,A -85,B 0,C 180,E1 -10354.423,E2 -10354.423} C_VEL
LIN {X 0,Y 410.194,Z 475.298,A -85,B 0,C 180,E1 -10355.407,E2 -10355.407} C_VEL
LIN {X 0,Y 410.396,Z 471.038,A -85,B 0,C 180,E1 -10356.662,E2 -10356.662} C_VEL
LIN {X 0,Y 410.639,Z 465.838,A -85,B 0,C 180,E1 -10357.869,E2 -10357.869} C_VEL
LIN {X 0,Y 410.962,Z 460.634,A -85,B 0,C 180,E1 -10358.853,E2 -10358.853} C_VEL
LIN {X 0,Y 411.421,Z 454.366,A -85,B 0,C 180,E1 -10359.835,E2 -10359.835} C_VEL
LIN {X 0,Y 411.866,Z 446.747,A -85,B 0,C 180,E1 -10360.818,E2 -10360.818} C_VEL
LIN {X 0,Y 412.398,Z 437.267,A -85,B 0,C 180,E1 -10361.8,E2 -10361.8} C_VEL
LIN {X 0,Y 412.964,Z 427.99,A -85,B 0,C 180,E1 -10362.532,E2 -10362.532} C_VEL
LIN {X 0,Y 413.365,Z 419.035,A -85,B 0,C 180,E1 -10363.081,E2 -10363.081} C_VEL
LIN {X 0,Y 413.706,Z 409.706,A -85,B 0,C 180,E1 -10363.508,E2 -10363.508} C_VEL
LIN {X 0,Y 413.981,Z 399.75,A -85,B 0,C 180,E1 -10363.814,E2 -10363.814} C_VEL
LIN {X 0,Y 414.394,Z 342.685,A -85,B 0,C 180,E1 -10364.826,E2 -10364.826} C_VEL
LIN {X 0,Y 411.447,Z 324.121,A -85,B 0,C 180,E1 -10365.288,E2 -10365.288} C_VEL
LIN {X 0,Y 411.419,Z 323.495,A -85,B 0,C 180,E1 -10365.353,E2 -10365.353} C_VEL
LIN {X 0,Y 412.053,Z 311.651,A -85,B 0,C 180,E1 -10368.393,E2 -10368.393} C_VEL
LIN {X 0,Y 412.507,Z 303.858,A -85,B 0,C 180,E1 -10370.438,E2 -10370.438} C_VEL
LIN {X 0,Y 411.938,Z 297.985,A -85,B 0,C 180,E1 -10372.045,E2 -10372.045} C_VEL
LIN {X 0,Y 411.262,Z 294.181,A -85,B 0,C 180,E1 -10373.143,E2 -10373.143} C_VEL
LIN {X 0,Y 411.17,Z 294.077,A -85,B 0,C 180,E1 -10376.385,E2 -10376.385} C_VEL
LIN {X 0,Y 411.195,Z 294.078,A -85,B 0,C 180,E1 -10379.712,E2 -10379.712} C_VEL
LIN {X 0,Y 411.202,Z 294.076,A -85,B 0,C 180,E1 -10383.155,E2 -10383.155} C_VEL
LIN {X 0,Y 411.188,Z 294.074,A -85,B 0,C 180,E1 -10386.551,E2 -10386.551} C_VEL
LIN {X 0,Y 411.165,Z 294.079,A -85,B 0,C 180,E1 -10389.72,E2 -10389.72} C_VEL
LIN {X 0,Y 411.157,Z 294.085,A -85,B 0,C 180,E1 -10393.134,E2 -10393.134} C_VEL
LIN {X 0,Y 411.158,Z 294.078,A -85,B 0,C 180,E1 -10395.881,E2 -10395.881} C_VEL
LIN {X 0,Y 411.157,Z 294.08,A -85,B 0,C 180,E1 -10399.493,E2 -10399.493} C_VEL
LIN {X 0,Y 411.181,Z 294.075,A -85,B 0,C 180,E1 -10402.025,E2 -10402.025} C_VEL
LIN {X 0,Y 411.196,Z 294.078,A -85,B 0,C 180,E1 -10405.123,E2 -10405.123} C_VEL
LIN {X 0,Y 411.155,Z 294.078,A -85,B 0,C 180,E1 -10408.002,E2 -10408.002} C_VEL
LIN {X 0,Y 411.164,Z 294.078,A -85,B 0,C 180,E1 -10411.406,E2 -10411.406} C_VEL
LIN {X 0,Y 411.18,Z 294.079,A -85,B 0,C 180,E1 -10414.941,E2 -10414.941} C_VEL
LIN {X 0,Y 411.193,Z 294.074,A -85,B 0,C 180,E1 -10417.913,E2 -10417.913} C_VEL
LIN {X 0,Y 411.201,Z 294.074,A -85,B 0,C 180,E1 -10421.05,E2 -10421.05} C_VEL
LIN {X 0,Y 411.2,Z 294.076,A -85,B 0,C 180,E1 -10424.129,E2 -10424.129} C_VEL
LIN {X 0,Y 411.294,Z 294.061,A -85,B 0,C 180,E1 -10427.165,E2 -10427.165} C_VEL
LIN {X 0,Y 411.279,Z 294.069,A -85,B 0,C 180,E1 -10430.161,E2 -10430.161} C_VEL
LIN {X 0,Y 411.381,Z 294.05,A -85,B 0,C 180,E1 -10433.132,E2 -10433.132} C_VEL
LIN {X 0,Y 411.278,Z 294.063,A -85,B 0,C 180,E1 -10435.099,E2 -10435.099} C_VEL
LIN {X 0,Y 411.491,Z 294.043,A -85,B 0,C 180,E1 -10438.042,E2 -10438.042} C_VEL
LIN {X 0,Y 411.365,Z 294.052,A -85,B 0,C 180,E1 -10440.979,E2 -10440.979} C_VEL
LIN {X 0,Y 411.415,Z 294.046,A -85,B 0,C 180,E1 -10442.937,E2 -10442.937} C_VEL
LIN {X 0,Y 411.417,Z 294.053,A -85,B 0,C 180,E1 -10445.883,E2 -10445.883} C_VEL
LIN {X 0,Y 411.296,Z 294.061,A -85,B 0,C 180,E1 -10448.846,E2 -10448.846} C_VEL
LIN {X 0,Y 411.263,Z 294.071,A -85,B 0,C 180,E1 -10451.833,E2 -10451.833} C_VEL
LIN {X 0,Y 411.22,Z 294.07,A -85,B 0,C 180,E1 -10454.854,E2 -10454.854} C_VEL
LIN {X 0,Y 411.204,Z 294.075,A -85,B 0,C 180,E1 -10457.917,E2 -10457.917} C_VEL
LIN {X 0,Y 411.183,Z 294.077,A -85,B 0,C 180,E1 -10461.035,E2 -10461.035} C_VEL
LIN {X 0,Y 411.18,Z 294.075,A -85,B 0,C 180,E1 -10464.218,E2 -10464.218} C_VEL
LIN {X 0,Y 411.138,Z 294.086,A -85,B 0,C 180,E1 -10467.486,E2 -10467.486} C_VEL
LIN {X 0,Y 411.187,Z 294.077,A -85,B 0,C 180,E1 -10469.714,E2 -10469.714} C_VEL
LIN {X 0,Y 411.197,Z 294.08,A -85,B 0,C 180,E1 -10473.157,E2 -10473.157} C_VEL
LIN {X 0,Y 411.184,Z 294.076,A -85,B 0,C 180,E1 -10476.553,E2 -10476.553} C_VEL
LIN {X 0,Y 411.162,Z 294.078,A -85,B 0,C 180,E1 -10479.721,E2 -10479.721} C_VEL
LIN {X 0,Y 411.155,Z 294.083,A -85,B 0,C 180,E1 -10483.136,E2 -10483.136} C_VEL
LIN {X 0,Y 411.158,Z 294.078,A -85,B 0,C 180,E1 -10485.882,E2 -10485.882} C_VEL
LIN {X 0,Y 411.152,Z 294.079,A -85,B 0,C 180,E1 -10489.493,E2 -10489.493} C_VEL
LIN {X 0,Y 411.179,Z 294.076,A -85,B 0,C 180,E1 -10492.026,E2 -10492.026} C_VEL
LIN {X 0,Y 411.198,Z 294.075,A -85,B 0,C 180,E1 -10495.124,E2 -10495.124} C_VEL
LIN {X 0,Y 411.16,Z 294.079,A -85,B 0,C 180,E1 -10498.003,E2 -10498.003} C_VEL
LIN {X 0,Y 411.169,Z 294.077,A -85,B 0,C 180,E1 -10501.407,E2 -10501.407} C_VEL
LIN {X 0,Y 411.185,Z 294.08,A -85,B 0,C 180,E1 -10504.942,E2 -10504.942} C_VEL
LIN {X 0,Y 411.291,Z 294.244,A -85,B 0,C 180,E1 -10506.93,E2 -10506.93} C_VEL
LIN {X 0,Y 412.42,Z 301.722,A -85,B 0,C 180,E1 -10509.032,E2 -10509.032} C_VEL
LIN {X 0,Y 412.288,Z 307.578,A -85,B 0,C 180,E1 -10510.586,E2 -10510.586} C_VEL
LIN {X 0,Y 411.498,Z 321.24,A -85,B 0,C 180,E1 -10514.142,E2 -10514.142} C_VEL
LIN {X 0,Y 411.417,Z 323.883,A -85,B 0,C 180,E1 -10514.742,E2 -10514.742} C_VEL
LIN {X 0,Y 413.597,Z 337.328,A -85,B 0,C 180,E1 -10515.095,E2 -10515.095} C_VEL
LIN {X 0,Y 414.436,Z 343.43,A -85,B 0,C 180,E1 -10515.233,E2 -10515.233} C_VEL
LIN {X 0,Y 414.026,Z 399.338,A -85,B 0,C 180,E1 -10516.222,E2 -10516.222} C_VEL
LIN {X 0,Y 413.714,Z 408.51,A -85,B 0,C 180,E1 -10516.492,E2 -10516.492} C_VEL
LIN {X 0,Y 413.426,Z 416.955,A -85,B 0,C 180,E1 -10516.858,E2 -10516.858} C_VEL
LIN {X 0,Y 413.042,Z 425.443,A -85,B 0,C 180,E1 -10517.346,E2 -10517.346} C_VEL
LIN {X 0,Y 412.649,Z 433.765,A -85,B 0,C 180,E1 -10517.958,E2 -10517.958} C_VEL
LIN {X 0,Y 412.189,Z 441.794,A -85,B 0,C 180,E1 -10518.692,E2 -10518.692} C_VEL
LIN {X 0,Y 411.621,Z 450.46,A -85,B 0,C 180,E1 -10519.673,E2 -10519.673} C_VEL
LIN {X 0,Y 411.054,Z 458.957,A -85,B 0,C 180,E1 -10520.901,E2 -10520.901} C_VEL
LIN {X 0,Y 410.648,Z 465.625,A -85,B 0,C 180,E1 -10522.131,E2 -10522.131} C_VEL
LIN {X 0,Y 410.435,Z 470.671,A -85,B 0,C 180,E1 -10523.289,E2 -10523.289} C_VEL
LIN {X 0,Y 410.213,Z 475.159,A -85,B 0,C 180,E1 -10524.593,E2 -10524.593} C_VEL
LIN {X 0,Y 409.99,Z 478.945,A -85,B 0,C 180,E1 -10526.068,E2 -10526.068} C_VEL
LIN {X 0,Y 409.949,Z 480.685,A -85,B 0,C 180,E1 -10527.052,E2 -10527.052} C_VEL
LIN {X 0,Y 409.968,Z 481.931,A -85,B 0,C 180,E1 -10528.035,E2 -10528.035} C_VEL
LIN {X 0,Y 409.917,Z 482.707,A -85,B 0,C 180,E1 -10529.018,E2 -10529.018} C_VEL
LIN {X 0,Y 409.885,Z 483,A -85,B 0,C 180,E1 -10530,E2 -10530} C_VEL
LIN {X 0,Y 409.917,Z 482.704,A -85,B 0,C 180,E1 -10530.982,E2 -10530.982} C_VEL
LIN {X 0,Y 409.968,Z 481.924,A -85,B 0,C 180,E1 -10531.965,E2 -10531.965} C_VEL
LIN {X 0,Y 409.949,Z 480.674,A -85,B 0,C 180,E1 -10532.948,E2 -10532.948} C_VEL
LIN {X 0,Y 410.053,Z 477.779,A -85,B 0,C 180,E1 -10534.423,E2 -10534.423} C_VEL
LIN {X 0,Y 410.212,Z 475.14,A -85,B 0,C 180,E1 -10535.407,E2 -10535.407} C_VEL
LIN {X 0,Y 410.435,Z 470.648,A -85,B 0,C 180,E1 -10536.71,E2 -10536.71} C_VEL
LIN {X 0,Y 410.644,Z 465.589,A -85,B 0,C 180,E1 -10537.869,E2 -10537.869} C_VEL
LIN {X 0,Y 411.054,Z 458.919,A -85,B 0,C 180,E1 -10539.099,E2 -10539.099} C_VEL
LIN {X 0,Y 411.62,Z 450.413,A -85,B 0,C 180,E1 -10540.327,E2 -10540.327} C_VEL
LIN {X 0,Y 412.182,Z 441.732,A -85,B 0,C 180,E1 -10541.308,E2 -10541.308} C_VEL
LIN {X 0,Y 412.661,Z 433.684,A -85,B 0,C 180,E1 -10542.042,E2 -10542.042} C_VEL
LIN {X 0,Y 413.066,Z 425.342,A -85,B 0,C 180,E1 -10542.653,E2 -10542.653} C_VEL
LIN {X 0,Y 413.423,Z 416.824,A -85,B 0,C 180,E1 -10543.142,E2 -10543.142} C_VEL
LIN {X 0,Y 413.787,Z 406.665,A -85,B 0,C 180,E1 -10543.568,E2 -10543.568} C_VEL
LIN {X 0,Y 414.053,Z 395.169,A -85,B 0,C 180,E1 -10543.867,E2 -10543.867} C_VEL
LIN {X 0,Y 414.319,Z 342.048,A -85,B 0,C 180,E1 -10544.788,E2 -10544.788} C_VEL
LIN {X 0,Y 411.454,Z 324.277,A -85,B 0,C 180,E1 -10545.224,E2 -10545.224} C_VEL
LIN {X 0,Y 411.409,Z 322.844,A -85,B 0,C 180,E1 -10545.442,E2 -10545.442} C_VEL
LIN {X 0,Y 412.169,Z 309.498,A -85,B 0,C 180,E1 -10548.903,E2 -10548.903} C_VEL
LIN {X 0,Y 412.493,Z 303.678,A -85,B 0,C 180,E1 -10550.433,E2 -10550.433} C_VEL
LIN {X 0,Y 411.718,Z 296.568,A -85,B 0,C 180,E1 -10552.386,E2 -10552.386} C_VEL
LIN {X 0,Y 411.258,Z 294.138,A -85,B 0,C 180,E1 -10553.144,E2 -10553.144} C_VEL
LIN {X 0,Y 411.169,Z 294.077,A -85,B 0,C 180,E1 -10556.385,E2 -10556.385} C_VEL
LIN {X 0,Y 411.193,Z 294.078,A -85,B 0,C 180,E1 -10559.713,E2 -10559.713} C_VEL
LIN {X 0,Y 411.201,Z 294.077,A -85,B 0,C 180,E1 -10563.155,E2 -10563.155} C_VEL
LIN {X 0,Y 411.187,Z 294.075,A -85,B 0,C 180,E1 -10566.552,E2 -10566.552} C_VEL
LIN {X 0,Y 411.164,Z 294.079,A -85,B 0,C 180,E1 -10569.72,E2 -10569.72} C_VEL
LIN {X 0,Y 411.156,Z 294.085,A -85,B 0,C 180,E1 -10573.135,E2 -10573.135} C_VEL
LIN {X 0,Y 411.157,Z 294.078,A -85,B 0,C 180,E1 -10575.881,E2 -10575.881} C_VEL
LIN {X 0,Y 411.151,Z 294.081,A -85,B 0,C 180,E1 -10579.492,E2 -10579.492} C_VEL
LIN {X 0,Y 411.178,Z 294.075,A -85,B 0,C 180,E1 -10582.025,E2 -10582.025} C_VEL
LIN {X 0,Y 411.195,Z 294.078,A -85,B 0,C 180,E1 -10585.123,E2 -10585.123} C_VEL
LIN {X 0,Y 411.155,Z 294.079,A -85,B 0,C 180,E1 -10588.002,E2 -10588.002} C_VEL
LIN {X 0,Y 411.163,Z 294.078,A -85,B 0,C 180,E1 -10591.406,E2 -10591.406} C_VEL
LIN {X 0,Y 411.179,Z 294.079,A -85,B 0,C 180,E1 -10594.941,E2 -10594.941} C_VEL
LIN {X 0,Y 411.192,Z 294.074,A -85,B 0,C 180,E1 -10597.913,E2 -10597.913} C_VEL
LIN {X 0,Y 411.201,Z 294.074,A -85,B 0,C 180,E1 -10601.05,E2 -10601.05} C_VEL
LIN {X 0,Y 411.199,Z 294.077,A -85,B 0,C 180,E1 -10604.13,E2 -10604.13} C_VEL
LIN {X 0,Y 411.293,Z 294.061,A -85,B 0,C 180,E1 -10607.165,E2 -10607.165} C_VEL
LIN {X 0,Y 411.277,Z 294.069,A -85,B 0,C 180,E1 -10610.161,E2 -10610.161} C_VEL
LIN {X 0,Y 411.38,Z 294.05,A -85,B 0,C 180,E1 -10613.132,E2 -10613.132} C_VEL
LIN {X 0,Y 411.278,Z 294.063,A -85,B 0,C 180,E1 -10615.099,E2 -10615.099} C_VEL
LIN {X 0,Y 411.491,Z 294.043,A -85,B 0,C 180,E1 -10618.043,E2 -10618.043} C_VEL
LIN {X 0,Y 411.366,Z 294.052,A -85,B 0,C 180,E1 -10620.979,E2 -10620.979} C_VEL
LIN {X 0,Y 411.416,Z 294.046,A -85,B 0,C 180,E1 -10622.938,E2 -10622.938} C_VEL
LIN {X 0,Y 411.381,Z 294.051,A -85,B 0,C 180,E1 -10626.45,E2 -10626.45} C_VEL
LIN {X 0,Y 411.295,Z 294.061,A -85,B 0,C 180,E1 -10628.847,E2 -10628.847} C_VEL
LIN {X 0,Y 411.263,Z 294.071,A -85,B 0,C 180,E1 -10631.833,E2 -10631.833} C_VEL
LIN {X 0,Y 411.219,Z 294.071,A -85,B 0,C 180,E1 -10634.854,E2 -10634.854} C_VEL
LIN {X 0,Y 411.198,Z 294.076,A -85,B 0,C 180,E1 -10637.918,E2 -10637.918} C_VEL
LIN {X 0,Y 411.183,Z 294.077,A -85,B 0,C 180,E1 -10641.035,E2 -10641.035} C_VEL
LIN {X 0,Y 411.181,Z 294.075,A -85,B 0,C 180,E1 -10644.218,E2 -10644.218} C_VEL
LIN {X 0,Y 411.138,Z 294.086,A -85,B 0,C 180,E1 -10647.487,E2 -10647.487} C_VEL
LIN {X 0,Y 411.186,Z 294.077,A -85,B 0,C 180,E1 -10649.714,E2 -10649.714} C_VEL
LIN {X 0,Y 411.197,Z 294.08,A -85,B 0,C 180,E1 -10653.157,E2 -10653.157} C_VEL
LIN {X 0,Y 411.184,Z 294.076,A -85,B 0,C 180,E1 -10656.553,E2 -10656.553} C_VEL
LIN {X 0,Y 411.162,Z 294.078,A -85,B 0,C 180,E1 -10659.721,E2 -10659.721} C_VEL
LIN {X 0,Y 411.156,Z 294.083,A -85,B 0,C 180,E1 -10663.136,E2 -10663.136} C_VEL
LIN {X 0,Y 411.159,Z 294.078,A -85,B 0,C 180,E1 -10665.883,E2 -10665.883} C_VEL
LIN {X 0,Y 411.153,Z 294.079,A -85,B 0,C 180,E1 -10669.494,E2 -10669.494} C_VEL
LIN {X 0,Y 411.18,Z 294.076,A -85,B 0,C 180,E1 -10672.026,E2 -10672.026} C_VEL
LIN {X 0,Y 411.199,Z 294.075,A -85,B 0,C 180,E1 -10675.124,E2 -10675.124} C_VEL
LIN {X 0,Y 411.157,Z 294.079,A -85,B 0,C 180,E1 -10678.003,E2 -10678.003} C_VEL
LIN {X 0,Y 411.166,Z 294.077,A -85,B 0,C 180,E1 -10681.407,E2 -10681.407} C_VEL
LIN {X 0,Y 411.186,Z 294.08,A -85,B 0,C 180,E1 -10684.942,E2 -10684.942} C_VEL
LIN {X 0,Y 411.303,Z 294.269,A -85,B 0,C 180,E1 -10686.996,E2 -10686.996} C_VEL
LIN {X 0,Y 412.353,Z 301.522,A -85,B 0,C 180,E1 -10689.028,E2 -10689.028} C_VEL
LIN {X 0,Y 412.29,Z 307.377,A -85,B 0,C 180,E1 -10690.586,E2 -10690.586} C_VEL
LIN {X 0,Y 411.5,Z 321.039,A -85,B 0,C 180,E1 -10694.142,E2 -10694.142} C_VEL
LIN {X 0,Y 411.4,Z 323.838,A -85,B 0,C 180,E1 -10694.789,E2 -10694.789} C_VEL
LIN {X 0,Y 412.694,Z 331.657,A -85,B 0,C 180,E1 -10695.014,E2 -10695.014} C_VEL
LIN {X 0,Y 414.435,Z 344.299,A -85,B 0,C 180,E1 -10695.3,E2 -10695.3} C_VEL
LIN {X 0,Y 413.997,Z 399.738,A -85,B 0,C 180,E1 -10696.283,E2 -10696.283} C_VEL
LIN {X 0,Y 413.716,Z 408.795,A -85,B 0,C 180,E1 -10696.555,E2 -10696.555} C_VEL
LIN {X 0,Y 413.348,Z 418.373,A -85,B 0,C 180,E1 -10696.981,E2 -10696.981} C_VEL
LIN {X 0,Y 412.898,Z 428.411,A -85,B 0,C 180,E1 -10697.591,E2 -10697.591} C_VEL
LIN {X 0,Y 412.389,Z 438.827,A -85,B 0,C 180,E1 -10698.449,E2 -10698.449} C_VEL
LIN {X 0,Y 411.846,Z 446.981,A -85,B 0,C 180,E1 -10699.305,E2 -10699.305} C_VEL
LIN {X 0,Y 411.424,Z 453.708,A -85,B 0,C 180,E1 -10700.165,E2 -10700.165} C_VEL
LIN {X 0,Y 410.973,Z 460.079,A -85,B 0,C 180,E1 -10701.147,E2 -10701.147} C_VEL
LIN {X 0,Y 410.619,Z 466.549,A -85,B 0,C 180,E1 -10702.378,E2 -10702.378} C_VEL
LIN {X 0,Y 410.436,Z 470.474,A -85,B 0,C 180,E1 -10703.29,E2 -10703.29} C_VEL
LIN {X 0,Y 410.214,Z 475.001,A -85,B 0,C 180,E1 -10704.593,E2 -10704.593} C_VEL
LIN {X 0,Y 410.055,Z 477.674,A -85,B 0,C 180,E1 -10705.577,E2 -10705.577} C_VEL
LIN {X 0,Y 409.951,Z 480.6,A -85,B 0,C 180,E1 -10707.052,E2 -10707.052} C_VEL
LIN {X 0,Y 409.969,Z 481.88,A -85,B 0,C 180,E1 -10708.035,E2 -10708.035} C_VEL
LIN {X 0,Y 409.892,Z 482.805,A -85,B 0,C 180,E1 -10709.385,E2 -10709.385} C_VEL
LIN {X 0,Y 409.194,Z 482.975,A -85,B 0,C 180,E1 -10710.206,E2 -10710.206} C_VEL
LIN {X 0,Y 406.312,Z 482.407,A -85,B 0,C 180,E1 -10711.537,E2 -10711.537} C_VEL
LIN {X 0,Y 403.478,Z 480.966,A -85,B 0,C 180,E1 -10712.875,E2 -10712.875} C_VEL
LIN {X 0,Y 402.877,Z 479.571,A -85,B 0,C 180,E1 -10713.695,E2 -10713.695} C_VEL
LIN {X 0,Y 403.056,Z 476.743,A -85,B 0,C 180,E1 -10715.001,E2 -10715.001} C_VEL
LIN {X 0,Y 403.191,Z 473.164,A -85,B 0,C 180,E1 -10716.205,E2 -10716.205} C_VEL
LIN {X 0,Y 403.54,Z 467.008,A -85,B 0,C 180,E1 -10717.757,E2 -10717.757} C_VEL
LIN {X 0,Y 403.845,Z 462.05,A -85,B 0,C 180,E1 -10718.758,E2 -10718.758} C_VEL
LIN {X 0,Y 404.292,Z 456.067,A -85,B 0,C 180,E1 -10719.758,E2 -10719.758} C_VEL
LIN {X 0,Y 404.765,Z 448.785,A -85,B 0,C 180,E1 -10720.757,E2 -10720.757} C_VEL
LIN {X 0,Y 405.261,Z 441.005,A -85,B 0,C 180,E1 -10721.63,E2 -10721.63} C_VEL
LIN {X 0,Y 405.71,Z 434.3,A -85,B 0,C 180,E1 -10722.251,E2 -10722.251} C_VEL
LIN {X 0,Y 406.112,Z 426.11,A -85,B 0,C 180,E1 -10722.874,E2 -10722.874} C_VEL
LIN {X 0,Y 406.515,Z 417.816,A -85,B 0,C 180,E1 -10723.369,E2 -10723.369} C_VEL
LIN {X 0,Y 406.814,Z 408.862,A -85,B 0,C 180,E1 -10723.773,E2 -10723.773} C_VEL
LIN {X 0,Y 407.098,Z 399.831,A -85,B 0,C 180,E1 -10724.05,E2 -10724.05} C_VEL
LIN {X 0,Y 407.466,Z 342.802,A -85,B 0,C 180,E1 -10725.082,E2 -10725.082} C_VEL
LIN {X 0,Y 404.456,Z 324.112,A -85,B 0,C 180,E1 -10725.559,E2 -10725.559} C_VEL
LIN {X 0,Y 404.398,Z 323.493,A -85,B 0,C 180,E1 -10725.626,E2 -10725.626} C_VEL
LIN {X 0,Y 405.108,Z 311.65,A -85,B 0,C 180,E1 -10728.72,E2 -10728.72} C_VEL
LIN {X 0,Y 405.465,Z 303.473,A -85,B 0,C 180,E1 -10730.913,E2 -10730.913} C_VEL
LIN {X 0,Y 404.454,Z 296.322,A -85,B 0,C 180,E1 -10732.934,E2 -10732.934} C_VEL
LIN {X 0,Y 404.226,Z 295.018,A -85,B 0,C 180,E1 -10733.38,E2 -10733.38} C_VEL
LIN {X 0,Y 404.115,Z 294.956,A -85,B 0,C 180,E1 -10736.882,E2 -10736.882} C_VEL
LIN {X 0,Y 404.142,Z 294.952,A -85,B 0,C 180,E1 -10740.285,E2 -10740.285} C_VEL
LIN {X 0,Y 404.135,Z 294.956,A -85,B 0,C 180,E1 -10743.812,E2 -10743.812} C_VEL
LIN {X 0,Y 404.131,Z 294.955,A -85,B 0,C 180,E1 -10746.874,E2 -10746.874} C_VEL
LIN {X 0,Y 404.113,Z 294.956,A -85,B 0,C 180,E1 -10750.074,E2 -10750.074} C_VEL
LIN {X 0,Y 404.137,Z 294.958,A -85,B 0,C 180,E1 -10753.081,E2 -10753.081} C_VEL
LIN {X 0,Y 404.115,Z 294.956,A -85,B 0,C 180,E1 -10755.921,E2 -10755.921} C_VEL
LIN {X 0,Y 404.097,Z 294.96,A -85,B 0,C 180,E1 -10758.632,E2 -10758.632} C_VEL
LIN {X 0,Y 404.136,Z 294.954,A -85,B 0,C 180,E1 -10761.494,E2 -10761.494} C_VEL
LIN {X 0,Y 404.167,Z 294.955,A -85,B 0,C 180,E1 -10764.982,E2 -10764.982} C_VEL
LIN {X 0,Y 404.13,Z 294.956,A -85,B 0,C 180,E1 -10768.442,E2 -10768.442} C_VEL
LIN {X 0,Y 404.141,Z 294.958,A -85,B 0,C 180,E1 -10770.862,E2 -10770.862} C_VEL
LIN {X 0,Y 404.144,Z 294.958,A -85,B 0,C 180,E1 -10774.722,E2 -10774.722} C_VEL
LIN {X 0,Y 404.157,Z 294.95,A -85,B 0,C 180,E1 -10777.507,E2 -10777.507} C_VEL
LIN {X 0,Y 404.147,Z 294.956,A -85,B 0,C 180,E1 -10780.707,E2 -10780.707} C_VEL
LIN {X 0,Y 404.17,Z 294.95,A -85,B 0,C 180,E1 -10783.846,E2 -10783.846} C_VEL
LIN {X 0,Y 404.275,Z 294.937,A -85,B 0,C 180,E1 -10786.938,E2 -10786.938} C_VEL
LIN {X 0,Y 404.245,Z 294.943,A -85,B 0,C 180,E1 -10789.988,E2 -10789.988} C_VEL
LIN {X 0,Y 404.331,Z 294.929,A -85,B 0,C 180,E1 -10793.011,E2 -10793.011} C_VEL
LIN {X 0,Y 404.25,Z 294.939,A -85,B 0,C 180,E1 -10795.013,E2 -10795.013} C_VEL
LIN {X 0,Y 404.46,Z 294.919,A -85,B 0,C 180,E1 -10798.008,E2 -10798.008} C_VEL
LIN {X 0,Y 404.336,Z 294.928,A -85,B 0,C 180,E1 -10800.996,E2 -10800.996} C_VEL
LIN {X 0,Y 404.349,Z 294.926,A -85,B 0,C 180,E1 -10802.989,E2 -10802.989} C_VEL
LIN {X 0,Y 404.366,Z 294.93,A -85,B 0,C 180,E1 -10805.986,E2 -10805.986} C_VEL
LIN {X 0,Y 404.245,Z 294.939,A -85,B 0,C 180,E1 -10809.002,E2 -10809.002} C_VEL
LIN {X 0,Y 404.238,Z 294.943,A -85,B 0,C 180,E1 -10812.042,E2 -10812.042} C_VEL
LIN {X 0,Y 404.165,Z 294.951,A -85,B 0,C 180,E1 -10815.119,E2 -10815.119} C_VEL
LIN {X 0,Y 404.156,Z 294.951,A -85,B 0,C 180,E1 -10818.24,E2 -10818.24} C_VEL
LIN {X 0,Y 404.125,Z 294.96,A -85,B 0,C 180,E1 -10821.42,E2 -10821.42} C_VEL
LIN {X 0,Y 404.126,Z 294.954,A -85,B 0,C 180,E1 -10824.669,E2 -10824.669} C_VEL
LIN {X 0,Y 404.094,Z 294.959,A -85,B 0,C 180,E1 -10828.007,E2 -10828.007} C_VEL
LIN {X 0,Y 404.134,Z 294.953,A -85,B 0,C 180,E1 -10830.286,E2 -10830.286} C_VEL
LIN {X 0,Y 404.13,Z 294.954,A -85,B 0,C 180,E1 -10833.814,E2 -10833.814} C_VEL
LIN {X 0,Y 404.127,Z 294.958,A -85,B 0,C 180,E1 -10836.875,E2 -10836.875} C_VEL
LIN {X 0,Y 404.11,Z 294.956,A -85,B 0,C 180,E1 -10840.075,E2 -10840.075} C_VEL
LIN {X 0,Y 404.135,Z 294.958,A -85,B 0,C 180,E1 -10843.082,E2 -10843.082} C_VEL
LIN {X 0,Y 404.114,Z 294.955,A -85,B 0,C 180,E1 -10845.923,E2 -10845.923} C_VEL
LIN {X 0,Y 404.096,Z 294.963,A -85,B 0,C 180,E1 -10848.633,E2 -10848.633} C_VEL
LIN {X 0,Y 404.134,Z 294.953,A -85,B 0,C 180,E1 -10851.496,E2 -10851.496} C_VEL
LIN {X 0,Y 404.173,Z 294.951,A -85,B 0,C 180,E1 -10854.984,E2 -10854.984} C_VEL
LIN {X 0,Y 404.134,Z 294.959,A -85,B 0,C 180,E1 -10858.443,E2 -10858.443} C_VEL
LIN {X 0,Y 404.146,Z 294.954,A -85,B 0,C 180,E1 -10860.863,E2 -10860.863} C_VEL
LIN {X 0,Y 404.15,Z 294.958,A -85,B 0,C 180,E1 -10864.723,E2 -10864.723} C_VEL
LIN {X 0,Y 404.215,Z 295.056,A -85,B 0,C 180,E1 -10866.716,E2 -10866.716} C_VEL
LIN {X 0,Y 405.294,Z 301.724,A -85,B 0,C 180,E1 -10868.645,E2 -10868.645} C_VEL
LIN {X 0,Y 405.384,Z 307.579,A -85,B 0,C 180,E1 -10870.241,E2 -10870.241} C_VEL
LIN {X 0,Y 404.533,Z 321.242,A -85,B 0,C 180,E1 -10873.861,E2 -10873.861} C_VEL
LIN {X 0,Y 404.434,Z 323.885,A -85,B 0,C 180,E1 -10874.472,E2 -10874.472} C_VEL
LIN {X 0,Y 406.848,Z 338.705,A -85,B 0,C 180,E1 -10874.866,E2 -10874.866} C_VEL
LIN {X 0,Y 407.569,Z 344.17,A -85,B 0,C 180,E1 -10874.991,E2 -10874.991} C_VEL
LIN {X 0,Y 407.154,Z 399.402,A -85,B 0,C 180,E1 -10875.986,E2 -10875.986} C_VEL
LIN {X 0,Y 406.837,Z 408.519,A -85,B 0,C 180,E1 -10876.26,E2 -10876.26} C_VEL
LIN {X 0,Y 406.525,Z 416.961,A -85,B 0,C 180,E1 -10876.631,E2 -10876.631} C_VEL
LIN {X 0,Y 406.129,Z 425.448,A -85,B 0,C 180,E1 -10877.127,E2 -10877.127} C_VEL
LIN {X 0,Y 405.698,Z 433.769,A -85,B 0,C 180,E1 -10877.748,E2 -10877.748} C_VEL
LIN {X 0,Y 405.226,Z 441.797,A -85,B 0,C 180,E1 -10878.496,E2 -10878.496} C_VEL
LIN {X 0,Y 404.653,Z 450.463,A -85,B 0,C 180,E1 -10879.493,E2 -10879.493} C_VEL
LIN {X 0,Y 404.045,Z 458.959,A -85,B 0,C 180,E1 -10880.741,E2 -10880.741} C_VEL
LIN {X 0,Y 403.619,Z 465.627,A -85,B 0,C 180,E1 -10881.993,E2 -10881.993} C_VEL
LIN {X 0,Y 403.412,Z 470.003,A -85,B 0,C 180,E1 -10882.996,E2 -10882.996} C_VEL
LIN {X 0,Y 403.185,Z 473.643,A -85,B 0,C 180,E1 -10883.997,E2 -10883.997} C_VEL
LIN {X 0,Y 403.085,Z 476.63,A -85,B 0,C 180,E1 -10884.999,E2 -10884.999} C_VEL
LIN {X 0,Y 402.912,Z 478.946,A -85,B 0,C 180,E1 -10885.999,E2 -10885.999} C_VEL
LIN {X 0,Y 402.85,Z 480.686,A -85,B 0,C 180,E1 -10887,E2 -10887} C_VEL
LIN {X 0,Y 402.866,Z 481.931,A -85,B 0,C 180,E1 -10888.001,E2 -10888.001} C_VEL
LIN {X 0,Y 402.845,Z 482.707,A -85,B 0,C 180,E1 -10889,E2 -10889} C_VEL
LIN {X 0,Y 402.812,Z 483,A -85,B 0,C 180,E1 -10890,E2 -10890} C_VEL
LIN {X 0,Y 402.845,Z 482.704,A -85,B 0,C 180,E1 -10891,E2 -10891} C_VEL
LIN {X 0,Y 402.866,Z 481.924,A -85,B 0,C 180,E1 -10891.999,E2 -10891.999} C_VEL
LIN {X 0,Y 402.85,Z 480.673,A -85,B 0,C 180,E1 -10893,E2 -10893} C_VEL
LIN {X 0,Y 402.986,Z 477.778,A -85,B 0,C 180,E1 -10894.501,E2 -10894.501} C_VEL
LIN {X 0,Y 403.139,Z 475.139,A -85,B 0,C 180,E1 -10895.502,E2 -10895.502} C_VEL
LIN {X 0,Y 403.35,Z 471.136,A -85,B 0,C 180,E1 -10896.7,E2 -10896.7} C_VEL
LIN {X 0,Y 403.542,Z 466.761,A -85,B 0,C 180,E1 -10897.757,E2 -10897.757} C_VEL
LIN {X 0,Y 403.852,Z 461.751,A -85,B 0,C 180,E1 -10898.758,E2 -10898.758} C_VEL
LIN {X 0,Y 404.293,Z 455.715,A -85,B 0,C 180,E1 -10899.758,E2 -10899.758} C_VEL
LIN {X 0,Y 404.781,Z 448.368,A -85,B 0,C 180,E1 -10900.757,E2 -10900.757} C_VEL
LIN {X 0,Y 405.3,Z 440.498,A -85,B 0,C 180,E1 -10901.629,E2 -10901.629} C_VEL
LIN {X 0,Y 405.779,Z 432.179,A -85,B 0,C 180,E1 -10902.376,E2 -10902.376} C_VEL
LIN {X 0,Y 406.312,Z 421.552,A -85,B 0,C 180,E1 -10903.122,E2 -10903.122} C_VEL
LIN {X 0,Y 406.759,Z 409.983,A -85,B 0,C 180,E1 -10903.679,E2 -10903.679} C_VEL
LIN {X 0,Y 407.077,Z 400.293,A -85,B 0,C 180,E1 -10903.987,E2 -10903.987} C_VEL
LIN {X 0,Y 407.501,Z 342.891,A -85,B 0,C 180,E1 -10905.026,E2 -10905.026} C_VEL
LIN {X 0,Y 404.453,Z 324.265,A -85,B 0,C 180,E1 -10905.494,E2 -10905.494} C_VEL
LIN {X 0,Y 404.403,Z 322.843,A -85,B 0,C 180,E1 -10905.717,E2 -10905.717} C_VEL
LIN {X 0,Y 405.22,Z 309.497,A -85,B 0,C 180,E1 -10909.24,E2 -10909.24} C_VEL
LIN {X 0,Y 405.436,Z 303.287,A -85,B 0,C 180,E1 -10910.911,E2 -10910.911} C_VEL
LIN {X 0,Y 404.427,Z 296.159,A -85,B 0,C 180,E1 -10912.925,E2 -10912.925} C_VEL
LIN {X 0,Y 404.213,Z 295.047,A -85,B 0,C 180,E1 -10913.281,E2 -10913.281} C_VEL
LIN {X 0,Y 404.114,Z 294.956,A -85,B 0,C 180,E1 -10916.882,E2 -10916.882} C_VEL
LIN {X 0,Y 404.139,Z 294.953,A -85,B 0,C 180,E1 -10920.285,E2 -10920.285} C_VEL
LIN {X 0,Y 404.134,Z 294.955,A -85,B 0,C 180,E1 -10923.812,E2 -10923.812} C_VEL
LIN {X 0,Y 404.13,Z 294.956,A -85,B 0,C 180,E1 -10926.874,E2 -10926.874} C_VEL
LIN {X 0,Y 404.112,Z 294.956,A -85,B 0,C 180,E1 -10930.074,E2 -10930.074} C_VEL
LIN {X 0,Y 404.136,Z 294.959,A -85,B 0,C 180,E1 -10933.081,E2 -10933.081} C_VEL
LIN {X 0,Y 404.114,Z 294.956,A -85,B 0,C 180,E1 -10935.922,E2 -10935.922} C_VEL
LIN {X 0,Y 404.095,Z 294.96,A -85,B 0,C 180,E1 -10938.632,E2 -10938.632} C_VEL
LIN {X 0,Y 404.133,Z 294.955,A -85,B 0,C 180,E1 -10941.494,E2 -10941.494} C_VEL
LIN {X 0,Y 404.166,Z 294.955,A -85,B 0,C 180,E1 -10944.982,E2 -10944.982} C_VEL
LIN {X 0,Y 404.129,Z 294.957,A -85,B 0,C 180,E1 -10948.442,E2 -10948.442} C_VEL
LIN {X 0,Y 404.141,Z 294.958,A -85,B 0,C 180,E1 -10950.862,E2 -10950.862} C_VEL
LIN {X 0,Y 404.144,Z 294.958,A -85,B 0,C 180,E1 -10954.723,E2 -10954.723} C_VEL
LIN {X 0,Y 404.156,Z 294.95,A -85,B 0,C 180,E1 -10957.507,E2 -10957.507} C_VEL
LIN {X 0,Y 404.147,Z 294.956,A -85,B 0,C 180,E1 -10960.707,E2 -10960.707} C_VEL
LIN {X 0,Y 404.17,Z 294.95,A -85,B 0,C 180,E1 -10963.846,E2 -10963.846} C_VEL
LIN {X 0,Y 404.274,Z 294.937,A -85,B 0,C 180,E1 -10966.939,E2 -10966.939} C_VEL
LIN {X 0,Y 404.243,Z 294.943,A -85,B 0,C 180,E1 -10969.988,E2 -10969.988} C_VEL
LIN {X 0,Y 404.33,Z 294.929,A -85,B 0,C 180,E1 -10973.011,E2 -10973.011} C_VEL
LIN {X 0,Y 404.249,Z 294.939,A -85,B 0,C 180,E1 -10975.013,E2 -10975.013} C_VEL
LIN {X 0,Y 404.46,Z 294.919,A -85,B 0,C 180,E1 -10978.009,E2 -10978.009} C_VEL
LIN {X 0,Y 404.336,Z 294.928,A -85,B 0,C 180,E1 -10980.996,E2 -10980.996} C_VEL
LIN {X 0,Y 404.349,Z 294.926,A -85,B 0,C 180,E1 -10982.989,E2 -10982.989} C_VEL
LIN {X 0,Y 404.334,Z 294.929,A -85,B 0,C 180,E1 -10986.445,E2 -10986.445} C_VEL
LIN {X 0,Y 404.245,Z 294.939,A -85,B 0,C 180,E1 -10989.002,E2 -10989.002} C_VEL
LIN {X 0,Y 404.238,Z 294.943,A -85,B 0,C 180,E1 -10992.042,E2 -10992.042} C_VEL
LIN {X 0,Y 404.164,Z 294.951,A -85,B 0,C 180,E1 -10995.12,E2 -10995.12} C_VEL
LIN {X 0,Y 404.152,Z 294.952,A -85,B 0,C 180,E1 -10998.241,E2 -10998.241} C_VEL
LIN {X 0,Y 404.126,Z 294.96,A -85,B 0,C 180,E1 -11001.42,E2 -11001.42} C_VEL
LIN {X 0,Y 404.126,Z 294.954,A -85,B 0,C 180,E1 -11004.669,E2 -11004.669} C_VEL
LIN {X 0,Y 404.095,Z 294.959,A -85,B 0,C 180,E1 -11008.007,E2 -11008.007} C_VEL
LIN {X 0,Y 404.133,Z 294.953,A -85,B 0,C 180,E1 -11010.286,E2 -11010.286} C_VEL
LIN {X 0,Y 404.131,Z 294.954,A -85,B 0,C 180,E1 -11013.814,E2 -11013.814} C_VEL
LIN {X 0,Y 404.127,Z 294.958,A -85,B 0,C 180,E1 -11016.875,E2 -11016.875} C_VEL
LIN {X 0,Y 404.111,Z 294.956,A -85,B 0,C 180,E1 -11020.076,E2 -11020.076} C_VEL
LIN {X 0,Y 404.136,Z 294.958,A -85,B 0,C 180,E1 -11023.083,E2 -11023.083} C_VEL
LIN {X 0,Y 404.116,Z 294.955,A -85,B 0,C 180,E1 -11025.923,E2 -11025.923} C_VEL
LIN {X 0,Y 404.097,Z 294.962,A -85,B 0,C 180,E1 -11028.633,E2 -11028.633} C_VEL
LIN {X 0,Y 404.135,Z 294.953,A -85,B 0,C 180,E1 -11031.496,E2 -11031.496} C_VEL
LIN {X 0,Y 404.174,Z 294.951,A -85,B 0,C 180,E1 -11034.984,E2 -11034.984} C_VEL
LIN {X 0,Y 404.131,Z 294.958,A -85,B 0,C 180,E1 -11038.444,E2 -11038.444} C_VEL
LIN {X 0,Y 404.145,Z 294.955,A -85,B 0,C 180,E1 -11040.863,E2 -11040.863} C_VEL
LIN {X 0,Y 404.151,Z 294.957,A -85,B 0,C 180,E1 -11044.723,E2 -11044.723} C_VEL
LIN {X 0,Y 404.235,Z 295.055,A -85,B 0,C 180,E1 -11046.774,E2 -11046.774} C_VEL
LIN {X 0,Y 405.415,Z 303.137,A -85,B 0,C 180,E1 -11049.092,E2 -11049.092} C_VEL
LIN {X 0,Y 405.222,Z 309.331,A -85,B 0,C 180,E1 -11050.76,E2 -11050.76} C_VEL
LIN {X 0,Y 404.469,Z 322.016,A -85,B 0,C 180,E1 -11054.118,E2 -11054.118} C_VEL
LIN {X 0,Y 404.404,Z 323.894,A -85,B 0,C 180,E1 -11054.524,E2 -11054.524} C_VEL
LIN {X 0,Y 406.98,Z 339.66,A -85,B 0,C 180,E1 -11054.941,E2 -11054.941} C_VEL
LIN {X 0,Y 407.576,Z 345.456,A -85,B 0,C 180,E1 -11055.068,E2 -11055.068} C_VEL
LIN {X 0,Y 407.11,Z 399.757,A -85,B 0,C 180,E1 -11056.046,E2 -11056.046} C_VEL
LIN {X 0,Y 406.838,Z 408.807,A -85,B 0,C 180,E1 -11056.323,E2 -11056.323} C_VEL
LIN {X 0,Y 406.448,Z 418.382,A -85,B 0,C 180,E1 -11056.756,E2 -11056.756} C_VEL
LIN {X 0,Y 405.982,Z 428.418,A -85,B 0,C 180,E1 -11057.376,E2 -11057.376} C_VEL
LIN {X 0,Y 405.44,Z 438.832,A -85,B 0,C 180,E1 -11058.248,E2 -11058.248} C_VEL
LIN {X 0,Y 404.864,Z 446.984,A -85,B 0,C 180,E1 -11059.119,E2 -11059.119} C_VEL
LIN {X 0,Y 404.412,Z 453.711,A -85,B 0,C 180,E1 -11059.992,E2 -11059.992} C_VEL
LIN {X 0,Y 403.954,Z 460.082,A -85,B 0,C 180,E1 -11060.992,E2 -11060.992} C_VEL
LIN {X 0,Y 403.567,Z 466.551,A -85,B 0,C 180,E1 -11062.244,E2 -11062.244} C_VEL
LIN {X 0,Y 403.351,Z 470.965,A -85,B 0,C 180,E1 -11063.3,E2 -11063.3} C_VEL
LIN {X 0,Y 403.141,Z 475.003,A -85,B 0,C 180,E1 -11064.498,E2 -11064.498} C_VEL
LIN {X 0,Y 402.989,Z 477.675,A -85,B 0,C 180,E1 -11065.499,E2 -11065.499} C_VEL
LIN {X 0,Y 402.851,Z 480.6,A -85,B 0,C 180,E1 -11067,E2 -11067} C_VEL
LIN {X 0,Y 402.867,Z 481.881,A -85,B 0,C 180,E1 -11068.001,E2 -11068.001} C_VEL
LIN {X 0,Y 402.819,Z 482.806,A -85,B 0,C 180,E1 -11069.379,E2 -11069.379} C_VEL
LIN {X 0,Y 402.813,Z 482.998,A -85,B 0,C 180,E1 -11070,E2 -11070} C_VEL
LIN {X 0,Y 402.845,Z 482.721,A -85,B 0,C 180,E1 -11071,E2 -11071} C_VEL
LIN {X 0,Y 402.848,Z 481.975,A -85,B 0,C 180,E1 -11071.999,E2 -11071.999} C_VEL
LIN {X 0,Y 402.877,Z 479.571,A -85,B 0,C 180,E1 -11073.695,E2 -11073.695} C_VEL
LIN {X 0,Y 402.305,Z 478.025,A -85,B 0,C 180,E1 -11074.504,E2 -11074.504} C_VEL
LIN {X 0,Y 399.643,Z 474.823,A -85,B 0,C 180,E1 -11075.793,E2 -11075.793} C_VEL
LIN {X 0,Y 396.998,Z 470.654,A -85,B 0,C 180,E1 -11077.038,E2 -11077.038} C_VEL
LIN {X 0,Y 396.46,Z 467.589,A -85,B 0,C 180,E1 -11077.769,E2 -11077.769} C_VEL
LIN {X 0,Y 396.818,Z 462.047,A -85,B 0,C 180,E1 -11078.915,E2 -11078.915} C_VEL
LIN {X 0,Y 397.293,Z 456.063,A -85,B 0,C 180,E1 -11079.932,E2 -11079.932} C_VEL
LIN {X 0,Y 397.788,Z 448.781,A -85,B 0,C 180,E1 -11080.948,E2 -11080.948} C_VEL
LIN {X 0,Y 398.304,Z 441,A -85,B 0,C 180,E1 -11081.836,E2 -11081.836} C_VEL
LIN {X 0,Y 398.781,Z 434.295,A -85,B 0,C 180,E1 -11082.467,E2 -11082.467} C_VEL
LIN {X 0,Y 399.205,Z 426.104,A -85,B 0,C 180,E1 -11083.1,E2 -11083.1} C_VEL
LIN {X 0,Y 399.628,Z 417.808,A -85,B 0,C 180,E1 -11083.604,E2 -11083.604} C_VEL
LIN {X 0,Y 399.936,Z 408.85,A -85,B 0,C 180,E1 -11084.015,E2 -11084.015} C_VEL
LIN {X 0,Y 400.221,Z 399.913,A -85,B 0,C 180,E1 -11084.294,E2 -11084.294} C_VEL
LIN {X 0,Y 400.644,Z 343.83,A -85,B 0,C 180,E1 -11085.326,E2 -11085.326} C_VEL
LIN {X 0,Y 397.471,Z 324.103,A -85,B 0,C 180,E1 -11085.84,E2 -11085.84} C_VEL
LIN {X 0,Y 397.452,Z 323.491,A -85,B 0,C 180,E1 -11085.906,E2 -11085.906} C_VEL
LIN {X 0,Y 398.283,Z 309.696,A -85,B 0,C 180,E1 -11089.588,E2 -11089.588} C_VEL
LIN {X 0,Y 398.398,Z 303.811,A -85,B 0,C 180,E1 -11091.208,E2 -11091.208} C_VEL
LIN {X 0,Y 397.191,Z 295.915,A -85,B 0,C 180,E1 -11093.538,E2 -11093.538} C_VEL
LIN {X 0,Y 397.084,Z 295.836,A -85,B 0,C 180,E1 -11097.398,E2 -11097.398} C_VEL
LIN {X 0,Y 397.097,Z 295.833,A -85,B 0,C 180,E1 -11099.862,E2 -11099.862} C_VEL
LIN {X 0,Y 397.109,Z 295.833,A -85,B 0,C 180,E1 -11103.273,E2 -11103.273} C_VEL
LIN {X 0,Y 397.102,Z 295.832,A -85,B 0,C 180,E1 -11105.734,E2 -11105.734} C_VEL
LIN {X 0,Y 397.089,Z 295.833,A -85,B 0,C 180,E1 -11108.854,E2 -11108.854} C_VEL
LIN {X 0,Y 397.05,Z 295.835,A -85,B 0,C 180,E1 -11112.268,E2 -11112.268} C_VEL
LIN {X 0,Y 397.081,Z 295.838,A -85,B 0,C 180,E1 -11115.068,E2 -11115.068} C_VEL
LIN {X 0,Y 397.046,Z 295.836,A -85,B 0,C 180,E1 -11118.023,E2 -11118.023} C_VEL
LIN {X 0,Y 397.087,Z 295.831,A -85,B 0,C 180,E1 -11121.723,E2 -11121.723} C_VEL
LIN {X 0,Y 397.11,Z 295.829,A -85,B 0,C 180,E1 -11125.505,E2 -11125.505} C_VEL
LIN {X 0,Y 397.068,Z 295.836,A -85,B 0,C 180,E1 -11129.117,E2 -11129.117} C_VEL
LIN {X 0,Y 397.054,Z 295.837,A -85,B 0,C 180,E1 -11132.251,E2 -11132.251} C_VEL
LIN {X 0,Y 397.094,Z 295.834,A -85,B 0,C 180,E1 -11134.864,E2 -11134.864} C_VEL
LIN {X 0,Y 397.085,Z 295.834,A -85,B 0,C 180,E1 -11138.181,E2 -11138.181} C_VEL
LIN {X 0,Y 397.101,Z 295.829,A -85,B 0,C 180,E1 -11141.423,E2 -11141.423} C_VEL
LIN {X 0,Y 397.114,Z 295.832,A -85,B 0,C 180,E1 -11144.605,E2 -11144.605} C_VEL
LIN {X 0,Y 397.209,Z 295.817,A -85,B 0,C 180,E1 -11147.741,E2 -11147.741} C_VEL
LIN {X 0,Y 397.225,Z 295.815,A -85,B 0,C 180,E1 -11150.837,E2 -11150.837} C_VEL
LIN {X 0,Y 397.318,Z 295.806,A -85,B 0,C 180,E1 -11153.908,E2 -11153.908} C_VEL
LIN {X 0,Y 397.429,Z 295.794,A -85,B 0,C 180,E1 -11157.973,E2 -11157.973} C_VEL
LIN {X 0,Y 397.427,Z 295.795,A -85,B 0,C 180,E1 -11162.027,E2 -11162.027} C_VEL
LIN {X 0,Y 397.317,Z 295.806,A -85,B 0,C 180,E1 -11166.092,E2 -11166.092} C_VEL
LIN {X 0,Y 397.217,Z 295.816,A -85,B 0,C 180,E1 -11169.163,E2 -11169.163} C_VEL
LIN {X 0,Y 397.204,Z 295.818,A -85,B 0,C 180,E1 -11172.258,E2 -11172.258} C_VEL
LIN {X 0,Y 397.114,Z 295.832,A -85,B 0,C 180,E1 -11175.394,E2 -11175.394} C_VEL
LIN {X 0,Y 397.104,Z 295.829,A -85,B 0,C 180,E1 -11178.576,E2 -11178.576} C_VEL
LIN {X 0,Y 397.083,Z 295.834,A -85,B 0,C 180,E1 -11181.819,E2 -11181.819} C_VEL
LIN {X 0,Y 397.094,Z 295.834,A -85,B 0,C 180,E1 -11185.136,E2 -11185.136} C_VEL
LIN {X 0,Y 397.054,Z 295.835,A -85,B 0,C 180,E1 -11188.549,E2 -11188.549} C_VEL
LIN {X 0,Y 397.071,Z 295.834,A -85,B 0,C 180,E1 -11191.836,E2 -11191.836} C_VEL
LIN {X 0,Y 397.109,Z 295.829,A -85,B 0,C 180,E1 -11194.495,E2 -11194.495} C_VEL
LIN {X 0,Y 397.085,Z 295.831,A -85,B 0,C 180,E1 -11198.277,E2 -11198.277} C_VEL
LIN {X 0,Y 397.044,Z 295.836,A -85,B 0,C 180,E1 -11201.977,E2 -11201.977} C_VEL
LIN {X 0,Y 397.08,Z 295.837,A -85,B 0,C 180,E1 -11205.07,E2 -11205.07} C_VEL
LIN {X 0,Y 397.046,Z 295.836,A -85,B 0,C 180,E1 -11208.024,E2 -11208.024} C_VEL
LIN {X 0,Y 397.086,Z 295.831,A -85,B 0,C 180,E1 -11211.724,E2 -11211.724} C_VEL
LIN {X 0,Y 397.115,Z 295.827,A -85,B 0,C 180,E1 -11215.507,E2 -11215.507} C_VEL
LIN {X 0,Y 397.072,Z 295.834,A -85,B 0,C 180,E1 -11219.118,E2 -11219.118} C_VEL
LIN {X 0,Y 397.059,Z 295.839,A -85,B 0,C 180,E1 -11222.252,E2 -11222.252} C_VEL
LIN {X 0,Y 397.128,Z 295.814,A -85,B 0,C 180,E1 -11225.982,E2 -11225.982} C_VEL
LIN {X 0,Y 397.227,Z 296.184,A -85,B 0,C 180,E1 -11226.629,E2 -11226.629} C_VEL
LIN {X 0,Y 398.39,Z 303.65,A -85,B 0,C 180,E1 -11228.792,E2 -11228.792} C_VEL
LIN {X 0,Y 398.292,Z 309.532,A -85,B 0,C 180,E1 -11230.412,E2 -11230.412} C_VEL
LIN {X 0,Y 397.485,Z 322.22,A -85,B 0,C 180,E1 -11233.831,E2 -11233.831} C_VEL
LIN {X 0,Y 397.418,Z 323.889,A -85,B 0,C 180,E1 -11234.191,E2 -11234.191} C_VEL
LIN {X 0,Y 399.887,Z 338.859,A -85,B 0,C 180,E1 -11234.599,E2 -11234.599} C_VEL
LIN {X 0,Y 400.695,Z 345.234,A -85,B 0,C 180,E1 -11234.747,E2 -11234.747} C_VEL
LIN {X 0,Y 400.278,Z 399.462,A -85,B 0,C 180,E1 -11235.742,E2 -11235.742} C_VEL
LIN {X 0,Y 399.955,Z 408.528,A -85,B 0,C 180,E1 -11236.018,E2 -11236.018} C_VEL
LIN {X 0,Y 399.624,Z 416.968,A -85,B 0,C 180,E1 -11236.396,E2 -11236.396} C_VEL
LIN {X 0,Y 399.226,Z 425.453,A -85,B 0,C 180,E1 -11236.9,E2 -11236.9} C_VEL
LIN {X 0,Y 398.763,Z 433.773,A -85,B 0,C 180,E1 -11237.532,E2 -11237.532} C_VEL
LIN {X 0,Y 398.28,Z 441.801,A -85,B 0,C 180,E1 -11238.292,E2 -11238.292} C_VEL
LIN {X 0,Y 397.73,Z 449.445,A -85,B 0,C 180,E1 -11239.179,E2 -11239.179} C_VEL
LIN {X 0,Y 397.153,Z 457.462,A -85,B 0,C 180,E1 -11240.322,E2 -11240.322} C_VEL
LIN {X 0,Y 396.674,Z 464.456,A -85,B 0,C 180,E1 -11241.595,E2 -11241.595} C_VEL
LIN {X 0,Y 396.374,Z 470.004,A -85,B 0,C 180,E1 -11242.871,E2 -11242.871} C_VEL
LIN {X 0,Y 396.069,Z 475.161,A -85,B 0,C 180,E1 -11244.399,E2 -11244.399} C_VEL
LIN {X 0,Y 395.838,Z 478.947,A -85,B 0,C 180,E1 -11245.928,E2 -11245.928} C_VEL
LIN {X 0,Y 395.754,Z 480.686,A -85,B 0,C 180,E1 -11246.946,E2 -11246.946} C_VEL
LIN {X 0,Y 395.764,Z 481.932,A -85,B 0,C 180,E1 -11247.965,E2 -11247.965} C_VEL
LIN {X 0,Y 395.757,Z 482.707,A -85,B 0,C 180,E1 -11248.982,E2 -11248.982} C_VEL
LIN {X 0,Y 395.723,Z 483,A -85,B 0,C 180,E1 -11250,E2 -11250} C_VEL
LIN {X 0,Y 395.757,Z 482.704,A -85,B 0,C 180,E1 -11251.018,E2 -11251.018} C_VEL
LIN {X 0,Y 395.764,Z 481.924,A -85,B 0,C 180,E1 -11252.035,E2 -11252.035} C_VEL
LIN {X 0,Y 395.754,Z 480.673,A -85,B 0,C 180,E1 -11253.054,E2 -11253.054} C_VEL
LIN {X 0,Y 395.921,Z 477.777,A -85,B 0,C 180,E1 -11254.582,E2 -11254.582} C_VEL
LIN {X 0,Y 396.068,Z 475.138,A -85,B 0,C 180,E1 -11255.601,E2 -11255.601} C_VEL
LIN {X 0,Y 396.309,Z 469.971,A -85,B 0,C 180,E1 -11257.131,E2 -11257.131} C_VEL
LIN {X 0,Y 396.734,Z 463.161,A -85,B 0,C 180,E1 -11258.66,E2 -11258.66} C_VEL
LIN {X 0,Y 397.287,Z 455.713,A -85,B 0,C 180,E1 -11259.932,E2 -11259.932} C_VEL
LIN {X 0,Y 397.796,Z 448.366,A -85,B 0,C 180,E1 -11260.948,E2 -11260.948} C_VEL
LIN {X 0,Y 398.351,Z 440.495,A -85,B 0,C 180,E1 -11261.835,E2 -11261.835} C_VEL
LIN {X 0,Y 398.862,Z 432.175,A -85,B 0,C 180,E1 -11262.594,E2 -11262.594} C_VEL
LIN {X 0,Y 399.421,Z 421.546,A -85,B 0,C 180,E1 -11263.352,E2 -11263.352} C_VEL
LIN {X 0,Y 399.869,Z 409.973,A -85,B 0,C 180,E1 -11263.92,E2 -11263.92} C_VEL
LIN {X 0,Y 400.197,Z 400.279,A -85,B 0,C 180,E1 -11264.232,E2 -11264.232} C_VEL
LIN {X 0,Y 400.571,Z 343.151,A -85,B 0,C 180,E1 -11265.287,E2 -11265.287} C_VEL
LIN {X 0,Y 397.46,Z 324.253,A -85,B 0,C 180,E1 -11265.774,E2 -11265.774} C_VEL
LIN {X 0,Y 397.453,Z 322.841,A -85,B 0,C 180,E1 -11265.999,E2 -11265.999} C_VEL
LIN {X 0,Y 398.29,Z 309.496,A -85,B 0,C 180,E1 -11269.588,E2 -11269.588} C_VEL
LIN {X 0,Y 398.467,Z 305.048,A -85,B 0,C 180,E1 -11270.806,E2 -11270.806} C_VEL
LIN {X 0,Y 397.861,Z 299.734,A -85,B 0,C 180,E1 -11272.32,E2 -11272.32} C_VEL
LIN {X 0,Y 397.174,Z 295.906,A -85,B 0,C 180,E1 -11273.502,E2 -11273.502} C_VEL
LIN {X 0,Y 397.083,Z 295.836,A -85,B 0,C 180,E1 -11277.398,E2 -11277.398} C_VEL
LIN {X 0,Y 397.095,Z 295.833,A -85,B 0,C 180,E1 -11279.862,E2 -11279.862} C_VEL
LIN {X 0,Y 397.108,Z 295.834,A -85,B 0,C 180,E1 -11283.273,E2 -11283.273} C_VEL
LIN {X 0,Y 397.101,Z 295.832,A -85,B 0,C 180,E1 -11285.734,E2 -11285.734} C_VEL
LIN {X 0,Y 397.088,Z 295.833,A -85,B 0,C 180,E1 -11288.854,E2 -11288.854} C_VEL
LIN {X 0,Y 397.048,Z 295.836,A -85,B 0,C 180,E1 -11292.269,E2 -11292.269} C_VEL
LIN {X 0,Y 397.08,Z 295.838,A -85,B 0,C 180,E1 -11295.068,E2 -11295.068} C_VEL
LIN {X 0,Y 397.045,Z 295.836,A -85,B 0,C 180,E1 -11298.023,E2 -11298.023} C_VEL
LIN {X 0,Y 397.085,Z 295.831,A -85,B 0,C 180,E1 -11301.723,E2 -11301.723} C_VEL
LIN {X 0,Y 397.109,Z 295.829,A -85,B 0,C 180,E1 -11305.505,E2 -11305.505} C_VEL
LIN {X 0,Y 397.068,Z 295.836,A -85,B 0,C 180,E1 -11309.117,E2 -11309.117} C_VEL
LIN {X 0,Y 397.053,Z 295.837,A -85,B 0,C 180,E1 -11312.251,E2 -11312.251} C_VEL
LIN {X 0,Y 397.094,Z 295.834,A -85,B 0,C 180,E1 -11314.864,E2 -11314.864} C_VEL
LIN {X 0,Y 397.084,Z 295.834,A -85,B 0,C 180,E1 -11318.181,E2 -11318.181} C_VEL
LIN {X 0,Y 397.1,Z 295.829,A -85,B 0,C 180,E1 -11321.424,E2 -11321.424} C_VEL
LIN {X 0,Y 397.113,Z 295.832,A -85,B 0,C 180,E1 -11324.605,E2 -11324.605} C_VEL
LIN {X 0,Y 397.209,Z 295.817,A -85,B 0,C 180,E1 -11327.742,E2 -11327.742} C_VEL
LIN {X 0,Y 397.224,Z 295.815,A -85,B 0,C 180,E1 -11330.838,E2 -11330.838} C_VEL
LIN {X 0,Y 397.318,Z 295.806,A -85,B 0,C 180,E1 -11333.908,E2 -11333.908} C_VEL
LIN {X 0,Y 397.429,Z 295.794,A -85,B 0,C 180,E1 -11337.973,E2 -11337.973} C_VEL
LIN {X 0,Y 397.427,Z 295.795,A -85,B 0,C 180,E1 -11342.027,E2 -11342.027} C_VEL
LIN {X 0,Y 397.292,Z 295.807,A -85,B 0,C 180,E1 -11346.437,E2 -11346.437} C_VEL
LIN {X 0,Y 397.216,Z 295.816,A -85,B 0,C 180,E1 -11349.163,E2 -11349.163} C_VEL
LIN {X 0,Y 397.204,Z 295.818,A -85,B 0,C 180,E1 -11352.259,E2 -11352.259} C_VEL
LIN {X 0,Y 397.113,Z 295.832,A -85,B 0,C 180,E1 -11355.395,E2 -11355.395} C_VEL
LIN {X 0,Y 397.101,Z 295.829,A -85,B 0,C 180,E1 -11358.577,E2 -11358.577} C_VEL
LIN {X 0,Y 397.084,Z 295.834,A -85,B 0,C 180,E1 -11361.819,E2 -11361.819} C_VEL
LIN {X 0,Y 397.094,Z 295.834,A -85,B 0,C 180,E1 -11365.136,E2 -11365.136} C_VEL
LIN {X 0,Y 397.054,Z 295.835,A -85,B 0,C 180,E1 -11368.549,E2 -11368.549} C_VEL
LIN {X 0,Y 397.07,Z 295.834,A -85,B 0,C 180,E1 -11371.836,E2 -11371.836} C_VEL
LIN {X 0,Y 397.11,Z 295.829,A -85,B 0,C 180,E1 -11374.495,E2 -11374.495} C_VEL
LIN {X 0,Y 397.084,Z 295.831,A -85,B 0,C 180,E1 -11378.277,E2 -11378.277} C_VEL
LIN {X 0,Y 397.045,Z 295.836,A -85,B 0,C 180,E1 -11381.977,E2 -11381.977} C_VEL
LIN {X 0,Y 397.081,Z 295.837,A -85,B 0,C 180,E1 -11385.07,E2 -11385.07} C_VEL
LIN {X 0,Y 397.047,Z 295.836,A -85,B 0,C 180,E1 -11388.025,E2 -11388.025} C_VEL
LIN {X 0,Y 397.087,Z 295.831,A -85,B 0,C 180,E1 -11391.724,E2 -11391.724} C_VEL
LIN {X 0,Y 397.116,Z 295.827,A -85,B 0,C 180,E1 -11395.507,E2 -11395.507} C_VEL
LIN {X 0,Y 397.07,Z 295.834,A -85,B 0,C 180,E1 -11399.118,E2 -11399.118} C_VEL
LIN {X 0,Y 397.058,Z 295.838,A -85,B 0,C 180,E1 -11402.253,E2 -11402.253} C_VEL
LIN {X 0,Y 397.129,Z 295.815,A -85,B 0,C 180,E1 -11405.982,E2 -11405.982} C_VEL
LIN {X 0,Y 397.185,Z 296.042,A -85,B 0,C 180,E1 -11406.632,E2 -11406.632} C_VEL
LIN {X 0,Y 398.36,Z 303.477,A -85,B 0,C 180,E1 -11408.798,E2 -11408.798} C_VEL
LIN {X 0,Y 398.292,Z 309.332,A -85,B 0,C 180,E1 -11410.412,E2 -11410.412} C_VEL
LIN {X 0,Y 397.425,Z 323.05,A -85,B 0,C 180,E1 -11414.092,E2 -11414.092} C_VEL
LIN {X 0,Y 397.463,Z 324.36,A -85,B 0,C 180,E1 -11414.274,E2 -11414.274} C_VEL
LIN {X 0,Y 400.61,Z 343.765,A -85,B 0,C 180,E1 -11414.77,E2 -11414.77} C_VEL
LIN {X 0,Y 400.237,Z 399.776,A -85,B 0,C 180,E1 -11415.802,E2 -11415.802} C_VEL
LIN {X 0,Y 399.958,Z 408.819,A -85,B 0,C 180,E1 -11416.083,E2 -11416.083} C_VEL
LIN {X 0,Y 399.564,Z 418.39,A -85,B 0,C 180,E1 -11416.523,E2 -11416.523} C_VEL
LIN {X 0,Y 399.075,Z 428.425,A -85,B 0,C 180,E1 -11417.154,E2 -11417.154} C_VEL
LIN {X 0,Y 398.497,Z 438.836,A -85,B 0,C 180,E1 -11418.04,E2 -11418.04} C_VEL
LIN {X 0,Y 397.899,Z 446.988,A -85,B 0,C 180,E1 -11418.926,E2 -11418.926} C_VEL
LIN {X 0,Y 397.411,Z 453.714,A -85,B 0,C 180,E1 -11419.814,E2 -11419.814} C_VEL
LIN {X 0,Y 396.925,Z 460.084,A -85,B 0,C 180,E1 -11420.831,E2 -11420.831} C_VEL
LIN {X 0,Y 396.539,Z 466.553,A -85,B 0,C 180,E1 -11422.105,E2 -11422.105} C_VEL
LIN {X 0,Y 396.272,Z 471.431,A -85,B 0,C 180,E1 -11423.304,E2 -11423.304} C_VEL
LIN {X 0,Y 396.006,Z 476.495,A -85,B 0,C 180,E1 -11424.909,E2 -11424.909} C_VEL
LIN {X 0,Y 395.841,Z 478.826,A -85,B 0,C 180,E1 -11425.928,E2 -11425.928} C_VEL
LIN {X 0,Y 395.755,Z 480.601,A -85,B 0,C 180,E1 -11426.946,E2 -11426.946} C_VEL
LIN {X 0,Y 395.765,Z 481.881,A -85,B 0,C 180,E1 -11427.965,E2 -11427.965} C_VEL
LIN {X 0,Y 395.758,Z 482.69,A -85,B 0,C 180,E1 -11428.982,E2 -11428.982} C_VEL
LIN {X 0,Y 395.725,Z 482.998,A -85,B 0,C 180,E1 -11430,E2 -11430} C_VEL
LIN {X 0,Y 395.757,Z 482.721,A -85,B 0,C 180,E1 -11431.018,E2 -11431.018} C_VEL
LIN {X 0,Y 395.746,Z 481.974,A -85,B 0,C 180,E1 -11432.035,E2 -11432.035} C_VEL
LIN {X 0,Y 395.792,Z 479.65,A -85,B 0,C 180,E1 -11433.714,E2 -11433.714} C_VEL
LIN {X 0,Y 395.978,Z 476.741,A -85,B 0,C 180,E1 -11435.091,E2 -11435.091} C_VEL
LIN {X 0,Y 396.232,Z 471.985,A -85,B 0,C 180,E1 -11436.646,E2 -11436.646} C_VEL
LIN {X 0,Y 396.46,Z 467.589,A -85,B 0,C 180,E1 -11437.769,E2 -11437.769} C_VEL
LIN {X 0,Y 395.963,Z 464.416,A -85,B 0,C 180,E1 -11438.475,E2 -11438.475} C_VEL
LIN {X 0,Y 393.549,Z 458.706,A -85,B 0,C 180,E1 -11439.6,E2 -11439.6} C_VEL
LIN {X 0,Y 391.215,Z 452.344,A -85,B 0,C 180,E1 -11440.658,E2 -11440.658} C_VEL
LIN {X 0,Y 390.854,Z 447.948,A -85,B 0,C 180,E1 -11441.252,E2 -11441.252} C_VEL
LIN {X 0,Y 391.343,Z 440.996,A -85,B 0,C 180,E1 -11442.05,E2 -11442.05} C_VEL
LIN {X 0,Y 391.866,Z 434.29,A -85,B 0,C 180,E1 -11442.691,E2 -11442.691} C_VEL
LIN {X 0,Y 392.308,Z 426.097,A -85,B 0,C 180,E1 -11443.335,E2 -11443.335} C_VEL
LIN {X 0,Y 392.74,Z 417.799,A -85,B 0,C 180,E1 -11443.847,E2 -11443.847} C_VEL
LIN {X 0,Y 393.065,Z 408.838,A -85,B 0,C 180,E1 -11444.265,E2 -11444.265} C_VEL
LIN {X 0,Y 393.354,Z 399.994,A -85,B 0,C 180,E1 -11444.547,E2 -11444.547} C_VEL
LIN {X 0,Y 393.779,Z 344.584,A -85,B 0,C 180,E1 -11445.585,E2 -11445.585} C_VEL
LIN {X 0,Y 390.515,Z 324.085,A -85,B 0,C 180,E1 -11446.13,E2 -11446.13} C_VEL
LIN {X 0,Y 390.457,Z 323.487,A -85,B 0,C 180,E1 -11446.2,E2 -11446.2} C_VEL
LIN {X 0,Y 391.207,Z 311.646,A -85,B 0,C 180,E1 -11449.411,E2 -11449.411} C_VEL
LIN {X 0,Y 391.466,Z 305.789,A -85,B 0,C 180,E1 -11451.042,E2 -11451.042} C_VEL
LIN {X 0,Y 390.354,Z 297.979,A -85,B 0,C 180,E1 -11453.333,E2 -11453.333} C_VEL
LIN {X 0,Y 390.125,Z 296.777,A -85,B 0,C 180,E1 -11453.77,E2 -11453.77} C_VEL
LIN {X 0,Y 390.04,Z 296.709,A -85,B 0,C 180,E1 -11456.773,E2 -11456.773} C_VEL
LIN {X 0,Y 390.035,Z 296.71,A -85,B 0,C 180,E1 -11460.299,E2 -11460.299} C_VEL
LIN {X 0,Y 390.066,Z 296.707,A -85,B 0,C 180,E1 -11464.024,E2 -11464.024} C_VEL
LIN {X 0,Y 390.036,Z 296.714,A -85,B 0,C 180,E1 -11467.549,E2 -11467.549} C_VEL
LIN {X 0,Y 390.012,Z 296.714,A -85,B 0,C 180,E1 -11470.814,E2 -11470.814} C_VEL
LIN {X 0,Y 390.039,Z 296.709,A -85,B 0,C 180,E1 -11473.884,E2 -11473.884} C_VEL
LIN {X 0,Y 390.041,Z 296.712,A -85,B 0,C 180,E1 -11476.787,E2 -11476.787} C_VEL
LIN {X 0,Y 390.004,Z 296.715,A -85,B 0,C 180,E1 -11479.554,E2 -11479.554} C_VEL
LIN {X 0,Y 390.034,Z 296.711,A -85,B 0,C 180,E1 -11482.449,E2 -11482.449} C_VEL
LIN {X 0,Y 390.055,Z 296.707,A -85,B 0,C 180,E1 -11486.044,E2 -11486.044} C_VEL
LIN {X 0,Y 390.035,Z 296.709,A -85,B 0,C 180,E1 -11489.87,E2 -11489.87} C_VEL
LIN {X 0,Y 390.022,Z 296.712,A -85,B 0,C 180,E1 -11493.225,E2 -11493.225} C_VEL
LIN {X 0,Y 390.051,Z 296.712,A -85,B 0,C 180,E1 -11496.766,E2 -11496.766} C_VEL
LIN {X 0,Y 390.076,Z 296.706,A -85,B 0,C 180,E1 -11499.981,E2 -11499.981} C_VEL
LIN {X 0,Y 390.097,Z 296.702,A -85,B 0,C 180,E1 -11503.246,E2 -11503.246} C_VEL
LIN {X 0,Y 390.187,Z 296.695,A -85,B 0,C 180,E1 -11506.561,E2 -11506.561} C_VEL
LIN {X 0,Y 390.156,Z 296.695,A -85,B 0,C 180,E1 -11509.622,E2 -11509.622} C_VEL
LIN {X 0,Y 390.236,Z 296.686,A -85,B 0,C 180,E1 -11512.757,E2 -11512.757} C_VEL
LIN {X 0,Y 390.193,Z 296.69,A -85,B 0,C 180,E1 -11514.833,E2 -11514.833} C_VEL
LIN {X 0,Y 390.396,Z 296.67,A -85,B 0,C 180,E1 -11517.937,E2 -11517.937} C_VEL
LIN {X 0,Y 390.393,Z 296.671,A -85,B 0,C 180,E1 -11522.063,E2 -11522.063} C_VEL
LIN {X 0,Y 390.272,Z 296.683,A -85,B 0,C 180,E1 -11526.203,E2 -11526.203} C_VEL
LIN {X 0,Y 390.175,Z 296.694,A -85,B 0,C 180,E1 -11529.329,E2 -11529.329} C_VEL
LIN {X 0,Y 390.186,Z 296.694,A -85,B 0,C 180,E1 -11533.439,E2 -11533.439} C_VEL
LIN {X 0,Y 390.098,Z 296.705,A -85,B 0,C 180,E1 -11537.288,E2 -11537.288} C_VEL
LIN {X 0,Y 390.063,Z 296.706,A -85,B 0,C 180,E1 -11540.464,E2 -11540.464} C_VEL
LIN {X 0,Y 390.048,Z 296.714,A -85,B 0,C 180,E1 -11543.353,E2 -11543.353} C_VEL
LIN {X 0,Y 390.021,Z 296.712,A -85,B 0,C 180,E1 -11546.775,E2 -11546.775} C_VEL
LIN {X 0,Y 390.028,Z 296.71,A -85,B 0,C 180,E1 -11550.301,E2 -11550.301} C_VEL
LIN {X 0,Y 390.062,Z 296.706,A -85,B 0,C 180,E1 -11554.025,E2 -11554.025} C_VEL
LIN {X 0,Y 390.031,Z 296.71,A -85,B 0,C 180,E1 -11557.781,E2 -11557.781} C_VEL
LIN {X 0,Y 390.009,Z 296.717,A -85,B 0,C 180,E1 -11560.815,E2 -11560.815} C_VEL
LIN {X 0,Y 390.038,Z 296.709,A -85,B 0,C 180,E1 -11563.885,E2 -11563.885} C_VEL
LIN {X 0,Y 390.041,Z 296.715,A -85,B 0,C 180,E1 -11566.789,E2 -11566.789} C_VEL
LIN {X 0,Y 390.004,Z 296.713,A -85,B 0,C 180,E1 -11569.555,E2 -11569.555} C_VEL
LIN {X 0,Y 390.034,Z 296.713,A -85,B 0,C 180,E1 -11572.451,E2 -11572.451} C_VEL
LIN {X 0,Y 390.065,Z 296.706,A -85,B 0,C 180,E1 -11575.976,E2 -11575.976} C_VEL
LIN {X 0,Y 390.039,Z 296.71,A -85,B 0,C 180,E1 -11579.871,E2 -11579.871} C_VEL
LIN {X 0,Y 390.027,Z 296.711,A -85,B 0,C 180,E1 -11583.226,E2 -11583.226} C_VEL
LIN {X 0,Y 390.154,Z 296.899,A -85,B 0,C 180,E1 -11586.373,E2 -11586.373} C_VEL
LIN {X 0,Y 391.274,Z 303.678,A -85,B 0,C 180,E1 -11588.395,E2 -11588.395} C_VEL
LIN {X 0,Y 391.496,Z 307.638,A -85,B 0,C 180,E1 -11589.525,E2 -11589.525} C_VEL
LIN {X 0,Y 390.685,Z 319.661,A -85,B 0,C 180,E1 -11592.836,E2 -11592.836} C_VEL
LIN {X 0,Y 390.456,Z 323.889,A -85,B 0,C 180,E1 -11593.901,E2 -11593.901} C_VEL
LIN {X 0,Y 393.335,Z 341.321,A -85,B 0,C 180,E1 -11594.381,E2 -11594.381} C_VEL
LIN {X 0,Y 393.847,Z 346.965,A -85,B 0,C 180,E1 -11594.507,E2 -11594.507} C_VEL
LIN {X 0,Y 393.419,Z 399.53,A -85,B 0,C 180,E1 -11595.489,E2 -11595.489} C_VEL
LIN {X 0,Y 393.076,Z 408.537,A -85,B 0,C 180,E1 -11595.769,E2 -11595.769} C_VEL
LIN {X 0,Y 392.739,Z 416.974,A -85,B 0,C 180,E1 -11596.153,E2 -11596.153} C_VEL
LIN {X 0,Y 392.335,Z 425.458,A -85,B 0,C 180,E1 -11596.666,E2 -11596.666} C_VEL
LIN {X 0,Y 391.84,Z 433.777,A -85,B 0,C 180,E1 -11597.308,E2 -11597.308} C_VEL
LIN {X 0,Y 391.315,Z 441.804,A -85,B 0,C 180,E1 -11598.081,E2 -11598.081} C_VEL
LIN {X 0,Y 390.703,Z 450.468,A -85,B 0,C 180,E1 -11599.113,E2 -11599.113} C_VEL
LIN {X 0,Y 390.021,Z 458.963,A -85,B 0,C 180,E1 -11600.405,E2 -11600.405} C_VEL
LIN {X 0,Y 389.529,Z 465.63,A -85,B 0,C 180,E1 -11601.701,E2 -11601.701} C_VEL
LIN {X 0,Y 389.243,Z 471.153,A -85,B 0,C 180,E1 -11603.052,E2 -11603.052} C_VEL
LIN {X 0,Y 388.979,Z 475.162,A -85,B 0,C 180,E1 -11604.297,E2 -11604.297} C_VEL
LIN {X 0,Y 388.861,Z 477.796,A -85,B 0,C 180,E1 -11605.335,E2 -11605.335} C_VEL
LIN {X 0,Y 388.662,Z 480.687,A -85,B 0,C 180,E1 -11606.89,E2 -11606.89} C_VEL
LIN {X 0,Y 388.663,Z 481.932,A -85,B 0,C 180,E1 -11607.927,E2 -11607.927} C_VEL
LIN {X 0,Y 388.657,Z 482.707,A -85,B 0,C 180,E1 -11608.964,E2 -11608.964} C_VEL
LIN {X 0,Y 388.638,Z 483,A -85,B 0,C 180,E1 -11610,E2 -11610} C_VEL
LIN {X 0,Y 388.657,Z 482.704,A -85,B 0,C 180,E1 -11611.036,E2 -11611.036} C_VEL
LIN {X 0,Y 388.662,Z 481.923,A -85,B 0,C 180,E1 -11612.073,E2 -11612.073} C_VEL
LIN {X 0,Y 388.662,Z 480.672,A -85,B 0,C 180,E1 -11613.11,E2 -11613.11} C_VEL
LIN {X 0,Y 388.856,Z 477.776,A -85,B 0,C 180,E1 -11614.665,E2 -11614.665} C_VEL
LIN {X 0,Y 388.978,Z 475.137,A -85,B 0,C 180,E1 -11615.703,E2 -11615.703} C_VEL
LIN {X 0,Y 389.202,Z 471.119,A -85,B 0,C 180,E1 -11616.948,E2 -11616.948} C_VEL
LIN {X 0,Y 389.448,Z 466.757,A -85,B 0,C 180,E1 -11618.039,E2 -11618.039} C_VEL
LIN {X 0,Y 389.804,Z 461.747,A -85,B 0,C 180,E1 -11619.077,E2 -11619.077} C_VEL
LIN {X 0,Y 390.272,Z 455.711,A -85,B 0,C 180,E1 -11620.112,E2 -11620.112} C_VEL
LIN {X 0,Y 390.815,Z 448.363,A -85,B 0,C 180,E1 -11621.146,E2 -11621.146} C_VEL
LIN {X 0,Y 391.401,Z 440.492,A -85,B 0,C 180,E1 -11622.048,E2 -11622.048} C_VEL
LIN {X 0,Y 391.944,Z 432.171,A -85,B 0,C 180,E1 -11622.82,E2 -11622.82} C_VEL
LIN {X 0,Y 392.528,Z 421.541,A -85,B 0,C 180,E1 -11623.591,E2 -11623.591} C_VEL
LIN {X 0,Y 393,Z 409.964,A -85,B 0,C 180,E1 -11624.168,E2 -11624.168} C_VEL
LIN {X 0,Y 393.332,Z 400.264,A -85,B 0,C 180,E1 -11624.486,E2 -11624.486} C_VEL
LIN {X 0,Y 393.854,Z 344.736,A -85,B 0,C 180,E1 -11625.525,E2 -11625.525} C_VEL
LIN {X 0,Y 390.503,Z 324.281,A -85,B 0,C 180,E1 -11626.061,E2 -11626.061} C_VEL
LIN {X 0,Y 390.468,Z 323.247,A -85,B 0,C 180,E1 -11626.199,E2 -11626.199} C_VEL
LIN {X 0,Y 391.364,Z 309.494,A -85,B 0,C 180,E1 -11629.949,E2 -11629.949} C_VEL
LIN {X 0,Y 391.27,Z 303.638,A -85,B 0,C 180,E1 -11631.605,E2 -11631.605} C_VEL
LIN {X 0,Y 390.127,Z 296.786,A -85,B 0,C 180,E1 -11633.7,E2 -11633.7} C_VEL
LIN {X 0,Y 390.038,Z 296.709,A -85,B 0,C 180,E1 -11636.773,E2 -11636.773} C_VEL
LIN {X 0,Y 390.033,Z 296.71,A -85,B 0,C 180,E1 -11640.299,E2 -11640.299} C_VEL
LIN {X 0,Y 390.065,Z 296.706,A -85,B 0,C 180,E1 -11644.024,E2 -11644.024} C_VEL
LIN {X 0,Y 390.035,Z 296.713,A -85,B 0,C 180,E1 -11647.549,E2 -11647.549} C_VEL
LIN {X 0,Y 390.011,Z 296.715,A -85,B 0,C 180,E1 -11650.814,E2 -11650.814} C_VEL
LIN {X 0,Y 390.038,Z 296.709,A -85,B 0,C 180,E1 -11653.884,E2 -11653.884} C_VEL
LIN {X 0,Y 390.04,Z 296.712,A -85,B 0,C 180,E1 -11656.787,E2 -11656.787} C_VEL
LIN {X 0,Y 390.003,Z 296.715,A -85,B 0,C 180,E1 -11659.554,E2 -11659.554} C_VEL
LIN {X 0,Y 390.032,Z 296.711,A -85,B 0,C 180,E1 -11662.45,E2 -11662.45} C_VEL
LIN {X 0,Y 390.054,Z 296.707,A -85,B 0,C 180,E1 -11666.044,E2 -11666.044} C_VEL
LIN {X 0,Y 390.034,Z 296.709,A -85,B 0,C 180,E1 -11669.87,E2 -11669.87} C_VEL
LIN {X 0,Y 390.021,Z 296.712,A -85,B 0,C 180,E1 -11673.225,E2 -11673.225} C_VEL
LIN {X 0,Y 390.05,Z 296.712,A -85,B 0,C 180,E1 -11676.767,E2 -11676.767} C_VEL
LIN {X 0,Y 390.076,Z 296.706,A -85,B 0,C 180,E1 -11679.982,E2 -11679.982} C_VEL
LIN {X 0,Y 390.096,Z 296.702,A -85,B 0,C 180,E1 -11683.246,E2 -11683.246} C_VEL
LIN {X 0,Y 390.186,Z 296.695,A -85,B 0,C 180,E1 -11686.561,E2 -11686.561} C_VEL
LIN {X 0,Y 390.155,Z 296.695,A -85,B 0,C 180,E1 -11689.623,E2 -11689.623} C_VEL
LIN {X 0,Y 390.236,Z 296.686,A -85,B 0,C 180,E1 -11692.758,E2 -11692.758} C_VEL
LIN {X 0,Y 390.192,Z 296.69,A -85,B 0,C 180,E1 -11694.833,E2 -11694.833} C_VEL
LIN {X 0,Y 390.396,Z 296.67,A -85,B 0,C 180,E1 -11697.937,E2 -11697.937} C_VEL
LIN {X 0,Y 390.393,Z 296.671,A -85,B 0,C 180,E1 -11702.063,E2 -11702.063} C_VEL
LIN {X 0,Y 390.253,Z 296.683,A -85,B 0,C 180,E1 -11706.427,E2 -11706.427} C_VEL
LIN {X 0,Y 390.175,Z 296.694,A -85,B 0,C 180,E1 -11709.33,E2 -11709.33} C_VEL
LIN {X 0,Y 390.187,Z 296.694,A -85,B 0,C 180,E1 -11713.439,E2 -11713.439} C_VEL
LIN {X 0,Y 390.098,Z 296.705,A -85,B 0,C 180,E1 -11717.288,E2 -11717.288} C_VEL
LIN {X 0,Y 390.043,Z 296.711,A -85,B 0,C 180,E1 -11721.123,E2 -11721.123} C_VEL
LIN {X 0,Y 390.033,Z 296.71,A -85,B 0,C 180,E1 -11724.484,E2 -11724.484} C_VEL
LIN {X 0,Y 390.008,Z 296.713,A -85,B 0,C 180,E1 -11727.998,E2 -11727.998} C_VEL
LIN {X 0,Y 390.012,Z 296.716,A -85,B 0,C 180,E1 -11731.506,E2 -11731.506} C_VEL
LIN {X 0,Y 390.062,Z 296.712,A -85,B 0,C 180,E1 -11735.209,E2 -11735.209} C_VEL
LIN {X 0,Y 390.051,Z 296.714,A -85,B 0,C 180,E1 -11739.097,E2 -11739.097} C_VEL
LIN {X 0,Y 390.024,Z 296.712,A -85,B 0,C 180,E1 -11742.373,E2 -11742.373} C_VEL
LIN {X 0,Y 390.036,Z 296.711,A -85,B 0,C 180,E1 -11745.355,E2 -11745.355} C_VEL
LIN {X 0,Y 390.01,Z 296.713,A -85,B 0,C 180,E1 -11748.185,E2 -11748.185} C_VEL
LIN {X 0,Y 390.053,Z 296.712,A -85,B 0,C 180,E1 -11750.904,E2 -11750.904} C_VEL
LIN {X 0,Y 390.078,Z 296.71,A -85,B 0,C 180,E1 -11754.793,E2 -11754.793} C_VEL
LIN {X 0,Y 390.016,Z 296.717,A -85,B 0,C 180,E1 -11758.496,E2 -11758.496} C_VEL
LIN {X 0,Y 390.013,Z 296.714,A -85,B 0,C 180,E1 -11762.004,E2 -11762.004} C_VEL
LIN {X 0,Y 390.055,Z 296.707,A -85,B 0,C 180,E1 -11765.518,E2 -11765.518} C_VEL
LIN {X 0,Y 390.164,Z 296.931,A -85,B 0,C 180,E1 -11766.444,E2 -11766.444} C_VEL
LIN {X 0,Y 391.236,Z 303.479,A -85,B 0,C 180,E1 -11768.393,E2 -11768.393} C_VEL
LIN {X 0,Y 391.367,Z 309.334,A -85,B 0,C 180,E1 -11770.051,E2 -11770.051} C_VEL
LIN {X 0,Y 390.459,Z 323.052,A -85,B 0,C 180,E1 -11773.8,E2 -11773.8} C_VEL
LIN {X 0,Y 390.446,Z 324.029,A -85,B 0,C 180,E1 -11773.968,E2 -11773.968} C_VEL
LIN {X 0,Y 393.8,Z 344.791,A -85,B 0,C 180,E1 -11774.519,E2 -11774.519} C_VEL
LIN {X 0,Y 393.37,Z 399.795,A -85,B 0,C 180,E1 -11775.548,E2 -11775.548} C_VEL
LIN {X 0,Y 393.08,Z 408.831,A -85,B 0,C 180,E1 -11775.835,E2 -11775.835} C_VEL
LIN {X 0,Y 392.678,Z 418.399,A -85,B 0,C 180,E1 -11776.282,E2 -11776.282} C_VEL
LIN {X 0,Y 392.175,Z 428.432,A -85,B 0,C 180,E1 -11776.924,E2 -11776.924} C_VEL
LIN {X 0,Y 391.532,Z 438.841,A -85,B 0,C 180,E1 -11777.824,E2 -11777.824} C_VEL
LIN {X 0,Y 390.934,Z 446.992,A -85,B 0,C 180,E1 -11778.726,E2 -11778.726} C_VEL
LIN {X 0,Y 390.424,Z 453.717,A -85,B 0,C 180,E1 -11779.63,E2 -11779.63} C_VEL
LIN {X 0,Y 389.918,Z 460.087,A -85,B 0,C 180,E1 -11780.665,E2 -11780.665} C_VEL
LIN {X 0,Y 389.487,Z 466.555,A -85,B 0,C 180,E1 -11781.961,E2 -11781.961} C_VEL
LIN {X 0,Y 389.18,Z 471.955,A -85,B 0,C 180,E1 -11783.324,E2 -11783.324} C_VEL
LIN {X 0,Y 388.93,Z 476.496,A -85,B 0,C 180,E1 -11784.816,E2 -11784.816} C_VEL
LIN {X 0,Y 388.771,Z 478.827,A -85,B 0,C 180,E1 -11785.853,E2 -11785.853} C_VEL
LIN {X 0,Y 388.664,Z 480.602,A -85,B 0,C 180,E1 -11786.89,E2 -11786.89} C_VEL
LIN {X 0,Y 388.664,Z 481.882,A -85,B 0,C 180,E1 -11787.927,E2 -11787.927} C_VEL
LIN {X 0,Y 388.658,Z 482.69,A -85,B 0,C 180,E1 -11788.964,E2 -11788.964} C_VEL
LIN {X 0,Y 388.639,Z 482.998,A -85,B 0,C 180,E1 -11790,E2 -11790} C_VEL
LIN {X 0,Y 388.656,Z 482.721,A -85,B 0,C 180,E1 -11791.036,E2 -11791.036} C_VEL
LIN {X 0,Y 388.645,Z 481.974,A -85,B 0,C 180,E1 -11792.073,E2 -11792.073} C_VEL
LIN {X 0,Y 388.656,Z 480.757,A -85,B 0,C 180,E1 -11793.11,E2 -11793.11} C_VEL
LIN {X 0,Y 388.854,Z 477.896,A -85,B 0,C 180,E1 -11794.665,E2 -11794.665} C_VEL
LIN {X 0,Y 388.963,Z 475.294,A -85,B 0,C 180,E1 -11795.703,E2 -11795.703} C_VEL
LIN {X 0,Y 389.208,Z 471.318,A -85,B 0,C 180,E1 -11796.948,E2 -11796.948} C_VEL
LIN {X 0,Y 389.504,Z 465.832,A -85,B 0,C 180,E1 -11798.299,E2 -11798.299} C_VEL
LIN {X 0,Y 389.909,Z 460.626,A -85,B 0,C 180,E1 -11799.336,E2 -11799.336} C_VEL
LIN {X 0,Y 390.406,Z 454.357,A -85,B 0,C 180,E1 -11800.371,E2 -11800.371} C_VEL
LIN {X 0,Y 390.854,Z 447.948,A -85,B 0,C 180,E1 -11801.252,E2 -11801.252} C_VEL
LIN {X 0,Y 390.496,Z 443.533,A -85,B 0,C 180,E1 -11801.807,E2 -11801.807} C_VEL
LIN {X 0,Y 388.238,Z 435.918,A -85,B 0,C 180,E1 -11802.667,E2 -11802.667} C_VEL
LIN {X 0,Y 386.169,Z 427.664,A -85,B 0,C 180,E1 -11803.443,E2 -11803.443} C_VEL
LIN {X 0,Y 385.629,Z 422.365,A -85,B 0,C 180,E1 -11803.838,E2 -11803.838} C_VEL
LIN {X 0,Y 386.167,Z 410.489,A -85,B 0,C 180,E1 -11804.458,E2 -11804.458} C_VEL
LIN {X 0,Y 386.471,Z 401.225,A -85,B 0,C 180,E1 -11804.779,E2 -11804.779} C_VEL
LIN {X 0,Y 386.752,Z 375.374,A -85,B 0,C 180,E1 -11805.294,E2 -11805.294} C_VEL
LIN {X 0,Y 386.923,Z 345.046,A -85,B 0,C 180,E1 -11805.859,E2 -11805.859} C_VEL
LIN {X 0,Y 383.536,Z 324.077,A -85,B 0,C 180,E1 -11806.432,E2 -11806.432} C_VEL
LIN {X 0,Y 383.511,Z 323.484,A -85,B 0,C 180,E1 -11806.501,E2 -11806.501} C_VEL
LIN {X 0,Y 384.275,Z 311.644,A -85,B 0,C 180,E1 -11809.776,E2 -11809.776} C_VEL
LIN {X 0,Y 384.37,Z 305.787,A -85,B 0,C 180,E1 -11811.449,E2 -11811.449} C_VEL
LIN {X 0,Y 383.086,Z 297.672,A -85,B 0,C 180,E1 -11813.947,E2 -11813.947} C_VEL
LIN {X 0,Y 382.98,Z 297.592,A -85,B 0,C 180,E1 -11817.307,E2 -11817.307} C_VEL
LIN {X 0,Y 382.98,Z 297.589,A -85,B 0,C 180,E1 -11820.918,E2 -11820.918} C_VEL
LIN {X 0,Y 383.014,Z 297.584,A -85,B 0,C 180,E1 -11824.667,E2 -11824.667} C_VEL
LIN {X 0,Y 382.99,Z 297.588,A -85,B 0,C 180,E1 -11827.902,E2 -11827.902} C_VEL
LIN {X 0,Y 382.956,Z 297.597,A -85,B 0,C 180,E1 -11831.35,E2 -11831.35} C_VEL
LIN {X 0,Y 382.984,Z 297.588,A -85,B 0,C 180,E1 -11834.301,E2 -11834.301} C_VEL
LIN {X 0,Y 382.991,Z 297.592,A -85,B 0,C 180,E1 -11837.237,E2 -11837.237} C_VEL
LIN {X 0,Y 382.981,Z 297.589,A -85,B 0,C 180,E1 -11840.418,E2 -11840.418} C_VEL
LIN {X 0,Y 383.008,Z 297.585,A -85,B 0,C 180,E1 -11844.042,E2 -11844.042} C_VEL
LIN {X 0,Y 382.978,Z 297.589,A -85,B 0,C 180,E1 -11847.578,E2 -11847.578} C_VEL
LIN {X 0,Y 382.968,Z 297.592,A -85,B 0,C 180,E1 -11850.298,E2 -11850.298} C_VEL
LIN {X 0,Y 382.995,Z 297.587,A -85,B 0,C 180,E1 -11854.044,E2 -11854.044} C_VEL
LIN {X 0,Y 382.977,Z 297.589,A -85,B 0,C 180,E1 -11857.333,E2 -11857.333} C_VEL
LIN {X 0,Y 383.023,Z 297.587,A -85,B 0,C 180,E1 -11860.714,E2 -11860.714} C_VEL
LIN {X 0,Y 383.009,Z 297.587,A -85,B 0,C 180,E1 -11864.023,E2 -11864.023} C_VEL
LIN {X 0,Y 383.127,Z 297.57,A -85,B 0,C 180,E1 -11867.283,E2 -11867.283} C_VEL
LIN {X 0,Y 383.133,Z 297.573,A -85,B 0,C 180,E1 -11870.497,E2 -11870.497} C_VEL
LIN {X 0,Y 383.229,Z 297.559,A -85,B 0,C 180,E1 -11873.683,E2 -11873.683} C_VEL
LIN {X 0,Y 383.362,Z 297.545,A -85,B 0,C 180,E1 -11877.899,E2 -11877.899} C_VEL
LIN {X 0,Y 383.358,Z 297.546,A -85,B 0,C 180,E1 -11882.101,E2 -11882.101} C_VEL
LIN {X 0,Y 383.228,Z 297.559,A -85,B 0,C 180,E1 -11886.317,E2 -11886.317} C_VEL
LIN {X 0,Y 383.126,Z 297.574,A -85,B 0,C 180,E1 -11889.503,E2 -11889.503} C_VEL
LIN {X 0,Y 383.117,Z 297.576,A -85,B 0,C 180,E1 -11893.536,E2 -11893.536} C_VEL
LIN {X 0,Y 383.044,Z 297.585,A -85,B 0,C 180,E1 -11897.434,E2 -11897.434} C_VEL
LIN {X 0,Y 383.007,Z 297.585,A -85,B 0,C 180,E1 -11900.642,E2 -11900.642} C_VEL
LIN {X 0,Y 382.998,Z 297.589,A -85,B 0,C 180,E1 -11903.809,E2 -11903.809} C_VEL
LIN {X 0,Y 382.96,Z 297.597,A -85,B 0,C 180,E1 -11907.309,E2 -11907.309} C_VEL
LIN {X 0,Y 382.973,Z 297.592,A -85,B 0,C 180,E1 -11910.919,E2 -11910.919} C_VEL
LIN {X 0,Y 383.004,Z 297.587,A -85,B 0,C 180,E1 -11914.669,E2 -11914.669} C_VEL
LIN {X 0,Y 382.986,Z 297.588,A -85,B 0,C 180,E1 -11917.903,E2 -11917.903} C_VEL
LIN {X 0,Y 382.954,Z 297.594,A -85,B 0,C 180,E1 -11921.351,E2 -11921.351} C_VEL
LIN {X 0,Y 382.983,Z 297.589,A -85,B 0,C 180,E1 -11924.303,E2 -11924.303} C_VEL
LIN {X 0,Y 382.976,Z 297.591,A -85,B 0,C 180,E1 -11927.237,E2 -11927.237} C_VEL
LIN {X 0,Y 382.98,Z 297.591,A -85,B 0,C 180,E1 -11930.42,E2 -11930.42} C_VEL
LIN {X 0,Y 383.018,Z 297.584,A -85,B 0,C 180,E1 -11934.045,E2 -11934.045} C_VEL
LIN {X 0,Y 382.981,Z 297.588,A -85,B 0,C 180,E1 -11937.579,E2 -11937.579} C_VEL
LIN {X 0,Y 382.972,Z 297.593,A -85,B 0,C 180,E1 -11940.299,E2 -11940.299} C_VEL
LIN {X 0,Y 383,Z 297.588,A -85,B 0,C 180,E1 -11944.046,E2 -11944.046} C_VEL
LIN {X 0,Y 383.104,Z 297.761,A -85,B 0,C 180,E1 -11946.162,E2 -11946.162} C_VEL
LIN {X 0,Y 384.364,Z 305.632,A -85,B 0,C 180,E1 -11948.55,E2 -11948.55} C_VEL
LIN {X 0,Y 384.434,Z 309.535,A -85,B 0,C 180,E1 -11949.675,E2 -11949.675} C_VEL
LIN {X 0,Y 383.51,Z 323.293,A -85,B 0,C 180,E1 -11953.499,E2 -11953.499} C_VEL
LIN {X 0,Y 383.51,Z 323.894,A -85,B 0,C 180,E1 -11953.601,E2 -11953.601} C_VEL
LIN {X 0,Y 385.978,Z 338.921,A -85,B 0,C 180,E1 -11954.03,E2 -11954.03} C_VEL
LIN {X 0,Y 387.031,Z 346.351,A -85,B 0,C 180,E1 -11954.215,E2 -11954.215} C_VEL
LIN {X 0,Y 386.55,Z 399.591,A -85,B 0,C 180,E1 -11955.227,E2 -11955.227} C_VEL
LIN {X 0,Y 386.21,Z 408.546,A -85,B 0,C 180,E1 -11955.51,E2 -11955.51} C_VEL
LIN {X 0,Y 385.873,Z 416.981,A -85,B 0,C 180,E1 -11955.901,E2 -11955.901} C_VEL
LIN {X 0,Y 385.445,Z 425.463,A -85,B 0,C 180,E1 -11956.423,E2 -11956.423} C_VEL
LIN {X 0,Y 384.924,Z 433.781,A -85,B 0,C 180,E1 -11957.076,E2 -11957.076} C_VEL
LIN {X 0,Y 384.351,Z 441.807,A -85,B 0,C 180,E1 -11957.861,E2 -11957.861} C_VEL
LIN {X 0,Y 383.734,Z 450.471,A -85,B 0,C 180,E1 -11958.913,E2 -11958.913} C_VEL
LIN {X 0,Y 383.023,Z 458.965,A -85,B 0,C 180,E1 -11960.228,E2 -11960.228} C_VEL
LIN {X 0,Y 382.509,Z 465.632,A -85,B 0,C 180,E1 -11961.548,E2 -11961.548} C_VEL
LIN {X 0,Y 382.265,Z 470.007,A -85,B 0,C 180,E1 -11962.606,E2 -11962.606} C_VEL
LIN {X 0,Y 381.974,Z 473.647,A -85,B 0,C 180,E1 -11963.662,E2 -11963.662} C_VEL
LIN {X 0,Y 381.852,Z 476.633,A -85,B 0,C 180,E1 -11964.72,E2 -11964.72} C_VEL
LIN {X 0,Y 381.702,Z 478.948,A -85,B 0,C 180,E1 -11965.776,E2 -11965.776} C_VEL
LIN {X 0,Y 381.574,Z 480.687,A -85,B 0,C 180,E1 -11966.833,E2 -11966.833} C_VEL
LIN {X 0,Y 381.561,Z 481.932,A -85,B 0,C 180,E1 -11967.889,E2 -11967.889} C_VEL
LIN {X 0,Y 381.556,Z 482.707,A -85,B 0,C 180,E1 -11968.945,E2 -11968.945} C_VEL
LIN {X 0,Y 381.538,Z 483,A -85,B 0,C 180,E1 -11970,E2 -11970} C_VEL
LIN {X 0,Y 381.556,Z 482.704,A -85,B 0,C 180,E1 -11971.055,E2 -11971.055} C_VEL
LIN {X 0,Y 381.561,Z 481.923,A -85,B 0,C 180,E1 -11972.111,E2 -11972.111} C_VEL
LIN {X 0,Y 381.574,Z 480.672,A -85,B 0,C 180,E1 -11973.167,E2 -11973.167} C_VEL
LIN {X 0,Y 381.793,Z 477.776,A -85,B 0,C 180,E1 -11974.751,E2 -11974.751} C_VEL
LIN {X 0,Y 381.891,Z 475.135,A -85,B 0,C 180,E1 -11975.809,E2 -11975.809} C_VEL
LIN {X 0,Y 382.104,Z 471.883,A -85,B 0,C 180,E1 -11976.866,E2 -11976.866} C_VEL
LIN {X 0,Y 382.41,Z 466.756,A -85,B 0,C 180,E1 -11978.188,E2 -11978.188} C_VEL
LIN {X 0,Y 382.775,Z 461.745,A -85,B 0,C 180,E1 -11979.245,E2 -11979.245} C_VEL
LIN {X 0,Y 383.266,Z 455.708,A -85,B 0,C 180,E1 -11980.299,E2 -11980.299} C_VEL
LIN {X 0,Y 383.862,Z 448.36,A -85,B 0,C 180,E1 -11981.351,E2 -11981.351} C_VEL
LIN {X 0,Y 384.445,Z 440.488,A -85,B 0,C 180,E1 -11982.269,E2 -11982.269} C_VEL
LIN {X 0,Y 385.031,Z 432.167,A -85,B 0,C 180,E1 -11983.054,E2 -11983.054} C_VEL
LIN {X 0,Y 385.644,Z 421.535,A -85,B 0,C 180,E1 -11983.838,E2 -11983.838} C_VEL
LIN {X 0,Y 386.14,Z 409.955,A -85,B 0,C 180,E1 -11984.425,E2 -11984.425} C_VEL
LIN {X 0,Y 386.486,Z 400.25,A -85,B 0,C 180,E1 -11984.748,E2 -11984.748} C_VEL
LIN {X 0,Y 387.05,Z 345.701,A -85,B 0,C 180,E1 -11985.786,E2 -11985.786} C_VEL
LIN {X 0,Y 383.541,Z 324.286,A -85,B 0,C 180,E1 -11986.36,E2 -11986.36} C_VEL
LIN {X 0,Y 383.51,Z 323.246,A -85,B 0,C 180,E1 -11986.501,E2 -11986.501} C_VEL
LIN {X 0,Y 384.282,Z 311.445,A -85,B 0,C 180,E1 -11989.775,E2 -11989.775} C_VEL
LIN {X 0,Y 384.362,Z 305.588,A -85,B 0,C 180,E1 -11991.45,E2 -11991.45} C_VEL
LIN {X 0,Y 383.088,Z 297.68,A -85,B 0,C 180,E1 -11993.875,E2 -11993.875} C_VEL
LIN {X 0,Y 382.978,Z 297.592,A -85,B 0,C 180,E1 -11997.307,E2 -11997.307} C_VEL
LIN {X 0,Y 382.978,Z 297.59,A -85,B 0,C 180,E1 -12000.918,E2 -12000.918} C_VEL
LIN {X 0,Y 383.013,Z 297.585,A -85,B 0,C 180,E1 -12004.668,E2 -12004.668} C_VEL
LIN {X 0,Y 382.989,Z 297.588,A -85,B 0,C 180,E1 -12007.902,E2 -12007.902} C_VEL
LIN {X 0,Y 382.955,Z 297.596,A -85,B 0,C 180,E1 -12011.35,E2 -12011.35} C_VEL
LIN {X 0,Y 382.983,Z 297.588,A -85,B 0,C 180,E1 -12014.302,E2 -12014.302} C_VEL
LIN {X 0,Y 382.976,Z 297.593,A -85,B 0,C 180,E1 -12017.236,E2 -12017.236} C_VEL
LIN {X 0,Y 382.979,Z 297.59,A -85,B 0,C 180,E1 -12020.418,E2 -12020.418} C_VEL
LIN {X 0,Y 383.007,Z 297.585,A -85,B 0,C 180,E1 -12024.043,E2 -12024.043} C_VEL
LIN {X 0,Y 382.977,Z 297.589,A -85,B 0,C 180,E1 -12027.578,E2 -12027.578} C_VEL
LIN {X 0,Y 382.967,Z 297.592,A -85,B 0,C 180,E1 -12030.298,E2 -12030.298} C_VEL
LIN {X 0,Y 382.994,Z 297.587,A -85,B 0,C 180,E1 -12034.045,E2 -12034.045} C_VEL
LIN {X 0,Y 382.977,Z 297.589,A -85,B 0,C 180,E1 -12037.333,E2 -12037.333} C_VEL
LIN {X 0,Y 383.022,Z 297.587,A -85,B 0,C 180,E1 -12040.714,E2 -12040.714} C_VEL
LIN {X 0,Y 383.009,Z 297.587,A -85,B 0,C 180,E1 -12044.024,E2 -12044.024} C_VEL
LIN {X 0,Y 383.127,Z 297.57,A -85,B 0,C 180,E1 -12047.284,E2 -12047.284} C_VEL
LIN {X 0,Y 383.132,Z 297.573,A -85,B 0,C 180,E1 -12050.498,E2 -12050.498} C_VEL
LIN {X 0,Y 383.229,Z 297.559,A -85,B 0,C 180,E1 -12053.683,E2 -12053.683} C_VEL
LIN {X 0,Y 383.362,Z 297.545,A -85,B 0,C 180,E1 -12057.899,E2 -12057.899} C_VEL
LIN {X 0,Y 383.358,Z 297.546,A -85,B 0,C 180,E1 -12062.101,E2 -12062.101} C_VEL
LIN {X 0,Y 383.22,Z 297.56,A -85,B 0,C 180,E1 -12066.413,E2 -12066.413} C_VEL
LIN {X 0,Y 383.126,Z 297.573,A -85,B 0,C 180,E1 -12069.503,E2 -12069.503} C_VEL
LIN {X 0,Y 383.117,Z 297.576,A -85,B 0,C 180,E1 -12073.536,E2 -12073.536} C_VEL
LIN {X 0,Y 383.044,Z 297.585,A -85,B 0,C 180,E1 -12077.434,E2 -12077.434} C_VEL
LIN {X 0,Y 383.008,Z 297.585,A -85,B 0,C 180,E1 -12080.642,E2 -12080.642} C_VEL
LIN {X 0,Y 382.999,Z 297.589,A -85,B 0,C 180,E1 -12083.81,E2 -12083.81} C_VEL
LIN {X 0,Y 382.961,Z 297.597,A -85,B 0,C 180,E1 -12087.309,E2 -12087.309} C_VEL
LIN {X 0,Y 382.972,Z 297.592,A -85,B 0,C 180,E1 -12090.92,E2 -12090.92} C_VEL
LIN {X 0,Y 383.005,Z 297.587,A -85,B 0,C 180,E1 -12094.669,E2 -12094.669} C_VEL
LIN {X 0,Y 382.987,Z 297.588,A -85,B 0,C 180,E1 -12097.903,E2 -12097.903} C_VEL
LIN {X 0,Y 382.955,Z 297.594,A -85,B 0,C 180,E1 -12101.351,E2 -12101.351} C_VEL
LIN {X 0,Y 382.984,Z 297.589,A -85,B 0,C 180,E1 -12104.303,E2 -12104.303} C_VEL
LIN {X 0,Y 382.977,Z 297.591,A -85,B 0,C 180,E1 -12107.237,E2 -12107.237} C_VEL
LIN {X 0,Y 382.982,Z 297.591,A -85,B 0,C 180,E1 -12110.42,E2 -12110.42} C_VEL
LIN {X 0,Y 383.019,Z 297.584,A -85,B 0,C 180,E1 -12114.045,E2 -12114.045} C_VEL
LIN {X 0,Y 382.98,Z 297.588,A -85,B 0,C 180,E1 -12117.58,E2 -12117.58} C_VEL
LIN {X 0,Y 382.971,Z 297.593,A -85,B 0,C 180,E1 -12120.299,E2 -12120.299} C_VEL
LIN {X 0,Y 383.001,Z 297.588,A -85,B 0,C 180,E1 -12124.046,E2 -12124.046} C_VEL
LIN {X 0,Y 383.101,Z 297.711,A -85,B 0,C 180,E1 -12126.198,E2 -12126.198} C_VEL
LIN {X 0,Y 384.341,Z 305.433,A -85,B 0,C 180,E1 -12128.549,E2 -12128.549} C_VEL
LIN {X 0,Y 384.43,Z 309.336,A -85,B 0,C 180,E1 -12129.675,E2 -12129.675} C_VEL
LIN {X 0,Y 383.511,Z 323.054,A -85,B 0,C 180,E1 -12133.499,E2 -12133.499} C_VEL
LIN {X 0,Y 383.496,Z 324.04,A -85,B 0,C 180,E1 -12133.669,E2 -12133.669} C_VEL
LIN {X 0,Y 387.001,Z 345.736,A -85,B 0,C 180,E1 -12134.257,E2 -12134.257} C_VEL
LIN {X 0,Y 386.502,Z 399.813,A -85,B 0,C 180,E1 -12135.286,E2 -12135.286} C_VEL
LIN {X 0,Y 386.212,Z 408.843,A -85,B 0,C 180,E1 -12135.578,E2 -12135.578} C_VEL
LIN {X 0,Y 385.792,Z 418.408,A -85,B 0,C 180,E1 -12136.033,E2 -12136.033} C_VEL
LIN {X 0,Y 385.28,Z 428.438,A -85,B 0,C 180,E1 -12136.686,E2 -12136.686} C_VEL
LIN {X 0,Y 384.579,Z 438.845,A -85,B 0,C 180,E1 -12137.601,E2 -12137.601} C_VEL
LIN {X 0,Y 383.979,Z 446.995,A -85,B 0,C 180,E1 -12138.519,E2 -12138.519} C_VEL
LIN {X 0,Y 383.452,Z 453.721,A -85,B 0,C 180,E1 -12139.439,E2 -12139.439} C_VEL
LIN {X 0,Y 382.916,Z 460.089,A -85,B 0,C 180,E1 -12140.492,E2 -12140.492} C_VEL
LIN {X 0,Y 382.456,Z 466.557,A -85,B 0,C 180,E1 -12141.813,E2 -12141.813} C_VEL
LIN {X 0,Y 382.142,Z 471.721,A -85,B 0,C 180,E1 -12143.135,E2 -12143.135} C_VEL
LIN {X 0,Y 381.854,Z 476.498,A -85,B 0,C 180,E1 -12144.72,E2 -12144.72} C_VEL
LIN {X 0,Y 381.704,Z 478.828,A -85,B 0,C 180,E1 -12145.777,E2 -12145.777} C_VEL
LIN {X 0,Y 381.576,Z 480.603,A -85,B 0,C 180,E1 -12146.833,E2 -12146.833} C_VEL
LIN {X 0,Y 381.562,Z 481.882,A -85,B 0,C 180,E1 -12147.889,E2 -12147.889} C_VEL
LIN {X 0,Y 381.557,Z 482.69,A -85,B 0,C 180,E1 -12148.945,E2 -12148.945} C_VEL
LIN {X 0,Y 381.54,Z 482.998,A -85,B 0,C 180,E1 -12150,E2 -12150} C_VEL
LIN {X 0,Y 381.555,Z 482.721,A -85,B 0,C 180,E1 -12151.055,E2 -12151.055} C_VEL
LIN {X 0,Y 381.544,Z 481.973,A -85,B 0,C 180,E1 -12152.111,E2 -12152.111} C_VEL
LIN {X 0,Y 381.568,Z 480.756,A -85,B 0,C 180,E1 -12153.167,E2 -12153.167} C_VEL
LIN {X 0,Y 381.79,Z 477.895,A -85,B 0,C 180,E1 -12154.751,E2 -12154.751} C_VEL
LIN {X 0,Y 381.877,Z 475.292,A -85,B 0,C 180,E1 -12155.809,E2 -12155.809} C_VEL
LIN {X 0,Y 382.106,Z 472.081,A -85,B 0,C 180,E1 -12156.866,E2 -12156.866} C_VEL
LIN {X 0,Y 382.4,Z 467.002,A -85,B 0,C 180,E1 -12158.189,E2 -12158.189} C_VEL
LIN {X 0,Y 382.775,Z 462.042,A -85,B 0,C 180,E1 -12159.245,E2 -12159.245} C_VEL
LIN {X 0,Y 383.282,Z 456.057,A -85,B 0,C 180,E1 -12160.298,E2 -12160.298} C_VEL
LIN {X 0,Y 383.856,Z 448.332,A -85,B 0,C 180,E1 -12161.409,E2 -12161.409} C_VEL
LIN {X 0,Y 384.391,Z 440.991,A -85,B 0,C 180,E1 -12162.271,E2 -12162.271} C_VEL
LIN {X 0,Y 385.042,Z 432.784,A -85,B 0,C 180,E1 -12163.054,E2 -12163.054} C_VEL
LIN {X 0,Y 385.535,Z 424.217,A -85,B 0,C 180,E1 -12163.708,E2 -12163.708} C_VEL
LIN {X 0,Y 385.629,Z 422.365,A -85,B 0,C 180,E1 -12163.838,E2 -12163.838} C_VEL
LIN {X 0,Y 385.143,Z 418.787,A -85,B 0,C 180,E1 -12164.098,E2 -12164.098} C_VEL
LIN {X 0,Y 382.597,Z 413.136,A -85,B 0,C 180,E1 -12164.513,E2 -12164.513} C_VEL
LIN {X 0,Y 380.044,Z 407.313,A -85,B 0,C 180,E1 -12164.855,E2 -12164.855} C_VEL
LIN {X 0,Y 379.53,Z 403.476,A -85,B 0,C 180,E1 -12164.995,E2 -12164.995} C_VEL
LIN {X 0,Y 379.794,Z 386.523,A -85,B 0,C 180,E1 -12165.367,E2 -12165.367} C_VEL
LIN {X 0,Y 380.106,Z 345.926,A -85,B 0,C 180,E1 -12166.134,E2 -12166.134} C_VEL
LIN {X 0,Y 376.574,Z 324.069,A -85,B 0,C 180,E1 -12166.745,E2 -12166.745} C_VEL
LIN {X 0,Y 376.598,Z 322.38,A -85,B 0,C 180,E1 -12167.093,E2 -12167.093} C_VEL
LIN {X 0,Y 377.364,Z 311.643,A -85,B 0,C 180,E1 -12170.153,E2 -12170.153} C_VEL
LIN {X 0,Y 377.431,Z 307.352,A -85,B 0,C 180,E1 -12171.403,E2 -12171.403} C_VEL
LIN {X 0,Y 376.126,Z 299.075,A -85,B 0,C 180,E1 -12173.942,E2 -12173.942} C_VEL
LIN {X 0,Y 376.017,Z 298.491,A -85,B 0,C 180,E1 -12174.279,E2 -12174.279} C_VEL
LIN {X 0,Y 375.924,Z 298.471,A -85,B 0,C 180,E1 -12177.864,E2 -12177.864} C_VEL
LIN {X 0,Y 375.955,Z 298.469,A -85,B 0,C 180,E1 -12181.561,E2 -12181.561} C_VEL
LIN {X 0,Y 375.953,Z 298.47,A -85,B 0,C 180,E1 -12185.415,E2 -12185.415} C_VEL
LIN {X 0,Y 375.932,Z 298.466,A -85,B 0,C 180,E1 -12188.262,E2 -12188.262} C_VEL
LIN {X 0,Y 375.909,Z 298.472,A -85,B 0,C 180,E1 -12191.596,E2 -12191.596} C_VEL
LIN {X 0,Y 375.916,Z 298.47,A -85,B 0,C 180,E1 -12194.729,E2 -12194.729} C_VEL
LIN {X 0,Y 375.911,Z 298.47,A -85,B 0,C 180,E1 -12197.697,E2 -12197.697} C_VEL
LIN {X 0,Y 375.93,Z 298.468,A -85,B 0,C 180,E1 -12200.533,E2 -12200.533} C_VEL
LIN {X 0,Y 375.952,Z 298.465,A -85,B 0,C 180,E1 -12203.496,E2 -12203.496} C_VEL
LIN {X 0,Y 375.951,Z 298.464,A -85,B 0,C 180,E1 -12205.887,E2 -12205.887} C_VEL
LIN {X 0,Y 375.954,Z 298.464,A -85,B 0,C 180,E1 -12209.686,E2 -12209.686} C_VEL
LIN {X 0,Y 375.91,Z 298.47,A -85,B 0,C 180,E1 -12212.134,E2 -12212.134} C_VEL
LIN {X 0,Y 375.928,Z 298.472,A -85,B 0,C 180,E1 -12214.533,E2 -12214.533} C_VEL
LIN {X 0,Y 375.962,Z 298.466,A -85,B 0,C 180,E1 -12216.886,E2 -12216.886} C_VEL
LIN {X 0,Y 375.965,Z 298.467,A -85,B 0,C 180,E1 -12220.337,E2 -12220.337} C_VEL
LIN {X 0,Y 375.965,Z 298.463,A -85,B 0,C 180,E1 -12223.716,E2 -12223.716} C_VEL
LIN {X 0,Y 376.095,Z 298.447,A -85,B 0,C 180,E1 -12227.042,E2 -12227.042} C_VEL
LIN {X 0,Y 376.103,Z 298.451,A -85,B 0,C 180,E1 -12230.318,E2 -12230.318} C_VEL
LIN {X 0,Y 376.188,Z 298.435,A -85,B 0,C 180,E1 -12233.564,E2 -12233.564} C_VEL
LIN {X 0,Y 376.327,Z 298.421,A -85,B 0,C 180,E1 -12237.859,E2 -12237.859} C_VEL
LIN {X 0,Y 376.322,Z 298.422,A -85,B 0,C 180,E1 -12242.14,E2 -12242.14} C_VEL
LIN {X 0,Y 376.187,Z 298.436,A -85,B 0,C 180,E1 -12246.436,E2 -12246.436} C_VEL
LIN {X 0,Y 376.097,Z 298.451,A -85,B 0,C 180,E1 -12249.682,E2 -12249.682} C_VEL
LIN {X 0,Y 376.081,Z 298.454,A -85,B 0,C 180,E1 -12253.657,E2 -12253.657} C_VEL
LIN {X 0,Y 375.998,Z 298.465,A -85,B 0,C 180,E1 -12257.589,E2 -12257.589} C_VEL
LIN {X 0,Y 375.971,Z 298.462,A -85,B 0,C 180,E1 -12260.832,E2 -12260.832} C_VEL
LIN {X 0,Y 375.926,Z 298.467,A -85,B 0,C 180,E1 -12264.286,E2 -12264.286} C_VEL
LIN {X 0,Y 375.903,Z 298.47,A -85,B 0,C 180,E1 -12266.661,E2 -12266.661} C_VEL
LIN {X 0,Y 375.905,Z 298.474,A -85,B 0,C 180,E1 -12269.085,E2 -12269.085} C_VEL
LIN {X 0,Y 375.948,Z 298.467,A -85,B 0,C 180,E1 -12271.563,E2 -12271.563} C_VEL
LIN {X 0,Y 375.942,Z 298.468,A -85,B 0,C 180,E1 -12275.417,E2 -12275.417} C_VEL
LIN {X 0,Y 375.929,Z 298.467,A -85,B 0,C 180,E1 -12278.263,E2 -12278.263} C_VEL
LIN {X 0,Y 375.907,Z 298.47,A -85,B 0,C 180,E1 -12281.597,E2 -12281.597} C_VEL
LIN {X 0,Y 375.915,Z 298.473,A -85,B 0,C 180,E1 -12284.731,E2 -12284.731} C_VEL
LIN {X 0,Y 375.902,Z 298.47,A -85,B 0,C 180,E1 -12287.697,E2 -12287.697} C_VEL
LIN {X 0,Y 375.93,Z 298.471,A -85,B 0,C 180,E1 -12290.534,E2 -12290.534} C_VEL
LIN {X 0,Y 375.957,Z 298.463,A -85,B 0,C 180,E1 -12293.497,E2 -12293.497} C_VEL
LIN {X 0,Y 375.955,Z 298.464,A -85,B 0,C 180,E1 -12295.889,E2 -12295.889} C_VEL
LIN {X 0,Y 375.958,Z 298.463,A -85,B 0,C 180,E1 -12299.688,E2 -12299.688} C_VEL
LIN {X 0,Y 375.914,Z 298.471,A -85,B 0,C 180,E1 -12302.135,E2 -12302.135} C_VEL
LIN {X 0,Y 376.031,Z 298.599,A -85,B 0,C 180,E1 -12305.931,E2 -12305.931} C_VEL
LIN {X 0,Y 377.238,Z 305.633,A -85,B 0,C 180,E1 -12308.124,E2 -12308.124} C_VEL
LIN {X 0,Y 377.486,Z 309.537,A -85,B 0,C 180,E1 -12309.284,E2 -12309.284} C_VEL
LIN {X 0,Y 376.603,Z 322.223,A -85,B 0,C 180,E1 -12312.908,E2 -12312.908} C_VEL
LIN {X 0,Y 376.55,Z 323.901,A -85,B 0,C 180,E1 -12313.289,E2 -12313.289} C_VEL
LIN {X 0,Y 379.134,Z 339.632,A -85,B 0,C 180,E1 -12313.747,E2 -12313.747} C_VEL
LIN {X 0,Y 380.217,Z 346.527,A -85,B 0,C 180,E1 -12313.927,E2 -12313.927} C_VEL
LIN {X 0,Y 379.705,Z 399.653,A -85,B 0,C 180,E1 -12314.955,E2 -12314.955} C_VEL
LIN {X 0,Y 379.31,Z 409.387,A -85,B 0,C 180,E1 -12315.275,E2 -12315.275} C_VEL
LIN {X 0,Y 378.897,Z 419.407,A -85,B 0,C 180,E1 -12315.773,E2 -12315.773} C_VEL
LIN {X 0,Y 378.191,Z 430.785,A -85,B 0,C 180,E1 -12316.568,E2 -12316.568} C_VEL
LIN {X 0,Y 377.583,Z 439.353,A -85,B 0,C 180,E1 -12317.367,E2 -12317.367} C_VEL
LIN {X 0,Y 377.002,Z 447.413,A -85,B 0,C 180,E1 -12318.304,E2 -12318.304} C_VEL
LIN {X 0,Y 376.461,Z 454.069,A -85,B 0,C 180,E1 -12319.241,E2 -12319.241} C_VEL
LIN {X 0,Y 375.885,Z 460.386,A -85,B 0,C 180,E1 -12320.313,E2 -12320.313} C_VEL
LIN {X 0,Y 375.47,Z 465.633,A -85,B 0,C 180,E1 -12321.388,E2 -12321.388} C_VEL
LIN {X 0,Y 375.187,Z 470.008,A -85,B 0,C 180,E1 -12322.466,E2 -12322.466} C_VEL
LIN {X 0,Y 374.836,Z 474.657,A -85,B 0,C 180,E1 -12323.9,E2 -12323.9} C_VEL
LIN {X 0,Y 374.717,Z 477.798,A -85,B 0,C 180,E1 -12325.159,E2 -12325.159} C_VEL
LIN {X 0,Y 374.49,Z 480.688,A -85,B 0,C 180,E1 -12326.773,E2 -12326.773} C_VEL
LIN {X 0,Y 374.46,Z 481.933,A -85,B 0,C 180,E1 -12327.849,E2 -12327.849} C_VEL
LIN {X 0,Y 374.456,Z 482.707,A -85,B 0,C 180,E1 -12328.925,E2 -12328.925} C_VEL
LIN {X 0,Y 374.439,Z 483,A -85,B 0,C 180,E1 -12330,E2 -12330} C_VEL
LIN {X 0,Y 374.456,Z 482.704,A -85,B 0,C 180,E1 -12331.075,E2 -12331.075} C_VEL
LIN {X 0,Y 374.46,Z 481.923,A -85,B 0,C 180,E1 -12332.151,E2 -12332.151} C_VEL
LIN {X 0,Y 374.49,Z 480.671,A -85,B 0,C 180,E1 -12333.227,E2 -12333.227} C_VEL
LIN {X 0,Y 374.711,Z 477.775,A -85,B 0,C 180,E1 -12334.841,E2 -12334.841} C_VEL
